gfCNCPoint1[27602] = {X 121.2453, Y 41.6137, Z -2.1667, A 0.000, B 0.000, C 0.000 }
gfCNCPoint1[27603] = {X 121.7141, Y 42.3988, Z -2.1667, A 0.000, B 0.000, C 0.000 }
gfCNCPoint1[27604] = {X 122.0072, Y 43.2649, Z -2.1667, A 0.000, B 0.000, C 0.000 }
gfCNCPoint1[27605] = {X 122.1114, Y 44.1734, Z -2.1667, A 0.000, B 0.000, C 0.000 }
gfCNCPoint1[27606] = {X 122.1116, Y 45.0000, Z -2.1667, A 0.000, B 0.000, C 0.000 }
gfCNCPoint1[27607] = {X 122.0033, Y 45.9613, Z -2.1667, A 0.000, B 0.000, C 0.000 }
gfCNCPoint1[27608] = {X 121.6838, Y 46.8744, Z -2.1667, A 0.000, B 0.000, C 0.000 }
gfCNCPoint1[27609] = {X 121.1691, Y 47.6935, Z -2.1667, A 0.000, B 0.000, C 0.000 }
gfCNCPoint1[27610] = {X 120.4850, Y 48.3775, Z -2.1667, A 0.000, B 0.000, C 0.000 }
gfCNCPoint1[27611] = {X 119.6660, Y 48.8922, Z -2.1667, A 0.000, B 0.000, C 0.000 }
gfCNCPoint1[27612] = {X 118.7529, Y 49.2117, Z -2.1667, A 0.000, B 0.000, C 0.000 }
gfCNCPoint1[27613] = {X 117.7916, Y 49.3200, Z -2.1667, A 0.000, B 0.000, C 0.000 }
gfCNCPoint1[27614] = {X 111.9185, Y 49.3200, Z -2.1667, A 0.000, B 0.000, C 0.000 }
gfCNCPoint1[27615] = {X 110.9619, Y 49.2128, Z -2.1667, A 0.000, B 0.000, C 0.000 }
gfCNCPoint1[27616] = {X 110.0529, Y 48.8964, Z -2.1667, A 0.000, B 0.000, C 0.000 }
gfCNCPoint1[27617] = {X 109.2365, Y 48.3866, Z -2.1667, A 0.000, B 0.000, C 0.000 }
gfCNCPoint1[27618] = {X 108.5532, Y 47.7087, Z -2.1667, A 0.000, B 0.000, C 0.000 }
gfCNCPoint1[27619] = {X 108.0369, Y 46.8963, Z -2.1667, A 0.000, B 0.000, C 0.000 }
gfCNCPoint1[27620] = {X 107.7134, Y 45.9898, Z -2.1667, A 0.000, B 0.000, C 0.000 }
gfCNCPoint1[27621] = {X 107.5986, Y 45.0341, Z -2.1667, A 0.000, B 0.000, C 0.000 }
gfCNCPoint1[27622] = {X 107.5985, Y 44.1778, Z -2.1667, A 0.000, B 0.000, C 0.000 }
gfCNCPoint1[27623] = {X 107.6341, Y 43.6353, Z -2.1667, A 0.000, B 0.000, C 0.000 }
gfCNCPoint1[27624] = {X 107.7405, Y 43.1023, Z -2.1667, A 0.000, B 0.000, C 0.000 }
gfCNCPoint1[27625] = {X 107.9071, Y 42.6088, Z -2.1667, A 0.000, B 0.000, C 0.000 }
gfCNCPoint1[27626] = {X 108.1343, Y 42.1400, Z -2.1667, A 0.000, B 0.000, C 0.000 }
gfCNCPoint1[27627] = {X 108.5859, Y 41.4664, Z -2.1667, A 0.000, B 0.000, C 0.000 }
gfCNCPoint1[27628] = {X 109.1269, Y 40.8623, Z -2.1667, A 0.000, B 0.000, C 0.000 }
gfCNCPoint1[27629] = {X 109.1268, Y 39.2937, Z -2.1667, A 0.000, B 0.000, C 0.000 }
gfCNCPoint1[27630] = {X 106.1118, Y 46.6615, Z -2.1667, A 0.000, B 0.000, C 0.000 }
gfCNCPoint1[27631] = {X 105.7417, Y 47.3611, Z -2.1667, A 0.000, B 0.000, C 0.000 }
gfCNCPoint1[27632] = {X 105.2502, Y 47.9815, Z -2.1667, A 0.000, B 0.000, C 0.000 }
gfCNCPoint1[27633] = {X 104.6538, Y 48.5018, Z -2.1667, A 0.000, B 0.000, C 0.000 }
gfCNCPoint1[27634] = {X 103.9724, Y 48.9046, Z -2.1667, A 0.000, B 0.000, C 0.000 }
gfCNCPoint1[27635] = {X 103.0287, Y 49.2242, Z -2.1667, A 0.000, B 0.000, C 0.000 }
gfCNCPoint1[27636] = {X 102.0368, Y 49.3191, Z -2.1667, A 0.000, B 0.000, C 0.000 }
gfCNCPoint1[27637] = {X 101.0496, Y 49.1842, Z -2.1667, A 0.000, B 0.000, C 0.000 }
gfCNCPoint1[27638] = {X 100.1195, Y 48.8268, Z -2.1667, A 0.000, B 0.000, C 0.000 }
gfCNCPoint1[27639] = {X 99.2961, Y 48.2657, Z -2.1667, A 0.000, B 0.000, C 0.000 }
gfCNCPoint1[27640] = {X 98.6231, Y 47.5309, Z -2.1667, A 0.000, B 0.000, C 0.000 }
gfCNCPoint1[27641] = {X 98.1363, Y 46.6615, Z -2.1667, A 0.000, B 0.000, C 0.000 }
gfCNCPoint1[27642] = {X 95.1301, Y 39.3093, Z -2.1667, A 0.000, B 0.000, C 0.000 }
gfCNCPoint1[27643] = {X 95.1302, Y 40.9055, Z -2.1667, A 0.000, B 0.000, C 0.000 }
gfCNCPoint1[27644] = {X 95.6600, Y 41.4488, Z -2.1667, A 0.000, B 0.000, C 0.000 }
gfCNCPoint1[27645] = {X 96.0887, Y 42.0749, Z -2.1667, A 0.000, B 0.000, C 0.000 }
gfCNCPoint1[27646] = {X 96.3308, Y 42.5747, Z -2.1667, A 0.000, B 0.000, C 0.000 }
gfCNCPoint1[27647] = {X 96.5082, Y 43.1009, Z -2.1667, A 0.000, B 0.000, C 0.000 }
gfCNCPoint1[27648] = {X 96.6185, Y 43.6488, Z -2.1667, A 0.000, B 0.000, C 0.000 }
gfCNCPoint1[27649] = {X 96.6585, Y 44.2063, Z -2.1667, A 0.000, B 0.000, C 0.000 }
gfCNCPoint1[27650] = {X 96.6583, Y 45.0415, Z -2.1667, A 0.000, B 0.000, C 0.000 }
gfCNCPoint1[27651] = {X 96.5422, Y 45.9960, Z -2.1667, A 0.000, B 0.000, C 0.000 }
gfCNCPoint1[27652] = {X 96.2178, Y 46.9011, Z -2.1667, A 0.000, B 0.000, C 0.000 }
gfCNCPoint1[27653] = {X 95.7012, Y 47.7120, Z -2.1667, A 0.000, B 0.000, C 0.000 }
gfCNCPoint1[27654] = {X 95.0181, Y 48.3886, Z -2.1667, A 0.000, B 0.000, C 0.000 }
gfCNCPoint1[27655] = {X 94.2022, Y 48.8973, Z -2.1667, A 0.000, B 0.000, C 0.000 }
gfCNCPoint1[27656] = {X 93.2940, Y 49.2130, Z -2.1667, A 0.000, B 0.000, C 0.000 }
gfCNCPoint1[27657] = {X 92.3385, Y 49.3200, Z -2.1667, A 0.000, B 0.000, C 0.000 }
gfCNCPoint1[27658] = {X 85.8951, Y 49.3200, Z -2.1667, A 0.000, B 0.000, C 0.000 }
gfCNCPoint1[27659] = {X 84.9387, Y 49.2128, Z -2.1667, A 0.000, B 0.000, C 0.000 }
gfCNCPoint1[27660] = {X 84.0297, Y 48.8965, Z -2.1667, A 0.000, B 0.000, C 0.000 }
gfCNCPoint1[27661] = {X 83.2134, Y 48.3869, Z -2.1667, A 0.000, B 0.000, C 0.000 }
gfCNCPoint1[27662] = {X 82.5301, Y 47.7091, Z -2.1667, A 0.000, B 0.000, C 0.000 }
gfCNCPoint1[27663] = {X 82.0138, Y 46.8970, Z -2.1667, A 0.000, B 0.000, C 0.000 }
gfCNCPoint1[27664] = {X 81.6902, Y 45.9906, Z -2.1667, A 0.000, B 0.000, C 0.000 }
gfCNCPoint1[27665] = {X 81.5752, Y 45.0351, Z -2.1667, A 0.000, B 0.000, C 0.000 }
gfCNCPoint1[27666] = {X 81.5751, Y 44.2068, Z -2.1667, A 0.000, B 0.000, C 0.000 }
gfCNCPoint1[27667] = {X 81.6809, Y 43.2777, Z -2.1667, A 0.000, B 0.000, C 0.000 }
gfCNCPoint1[27668] = {X 81.9815, Y 42.3922, Z -2.1667, A 0.000, B 0.000, C 0.000 }
gfCNCPoint1[27669] = {X 82.4630, Y 41.5906, Z -2.1667, A 0.000, B 0.000, C 0.000 }
gfCNCPoint1[27670] = {X 83.1037, Y 40.9095, Z -2.1667, A 0.000, B 0.000, C 0.000 }
gfCNCPoint1[27671] = {X 83.1036, Y 28.5922, Z -2.1667, A 0.000, B 0.000, C 0.000 }
gfCNCPoint1[27672] = {X 79.1036, Y 28.5922, Z -2.1667, A 0.000, B 0.000, C 0.000 }
gfCNCPoint1[27673] = {X 83.1836, Y 28.5922, Z -2.1667, A 0.000, B 0.000, C 0.000 }
gfCNCPoint1[27674] = {X 83.1834, Y 16.2375, Z -2.1667, A 0.000, B 0.000, C 0.000 }
gfCNCPoint1[27675] = {X 82.5450, Y 15.5770, Z -2.1667, A 0.000, B 0.000, C 0.000 }
gfCNCPoint1[27676] = {X 82.0638, Y 14.7944, Z -2.1667, A 0.000, B 0.000, C 0.000 }
gfCNCPoint1[27677] = {X 81.7625, Y 13.9265, Z -2.1667, A 0.000, B 0.000, C 0.000 }
gfCNCPoint1[27678] = {X 81.6552, Y 13.0142, Z -2.1667, A 0.000, B 0.000, C 0.000 }
gfCNCPoint1[27679] = {X 81.6551, Y 12.1868, Z -2.1667, A 0.000, B 0.000, C 0.000 }
gfCNCPoint1[27680] = {X 81.7614, Y 11.2433, Z -2.1667, A 0.000, B 0.000, C 0.000 }
gfCNCPoint1[27681] = {X 82.0750, Y 10.3472, Z -2.1667, A 0.000, B 0.000, C 0.000 }
gfCNCPoint1[27682] = {X 82.5801, Y 9.5432, Z -2.1667, A 0.000, B 0.000, C 0.000 }
gfCNCPoint1[27683] = {X 83.2515, Y 8.8719, Z -2.1667, A 0.000, B 0.000, C 0.000 }
gfCNCPoint1[27684] = {X 84.0554, Y 8.3667, Z -2.1667, A 0.000, B 0.000, C 0.000 }
gfCNCPoint1[27685] = {X 84.9516, Y 8.0531, Z -2.1667, A 0.000, B 0.000, C 0.000 }
gfCNCPoint1[27686] = {X 85.8951, Y 7.9468, Z -2.1667, A 0.000, B 0.000, C 0.000 }
gfCNCPoint1[27687] = {X 94.0497, Y 7.9468, Z -2.1667, A 0.000, B 0.000, C 0.000 }
gfCNCPoint1[27688] = {X 94.9932, Y 8.0531, Z -2.1667, A 0.000, B 0.000, C 0.000 }
gfCNCPoint1[27689] = {X 95.8893, Y 8.3667, Z -2.1667, A 0.000, B 0.000, C 0.000 }
gfCNCPoint1[27690] = {X 96.6933, Y 8.8718, Z -2.1667, A 0.000, B 0.000, C 0.000 }
gfCNCPoint1[27691] = {X 97.3646, Y 9.5432, Z -2.1667, A 0.000, B 0.000, C 0.000 }
gfCNCPoint1[27692] = {X 97.8698, Y 10.3471, Z -2.1667, A 0.000, B 0.000, C 0.000 }
gfCNCPoint1[27693] = {X 98.1834, Y 11.2433, Z -2.1667, A 0.000, B 0.000, C 0.000 }
gfCNCPoint1[27694] = {X 98.2897, Y 12.1868, Z -2.1667, A 0.000, B 0.000, C 0.000 }
gfCNCPoint1[27695] = {X 98.2897, Y 12.9781, Z -2.1667, A 0.000, B 0.000, C 0.000 }
gfCNCPoint1[27696] = {X 98.2155, Y 13.7669, Z -2.1667, A 0.000, B 0.000, C 0.000 }
gfCNCPoint1[27697] = {X 97.9959, Y 14.5281, Z -2.1667, A 0.000, B 0.000, C 0.000 }
gfCNCPoint1[27698] = {X 97.6385, Y 15.2352, Z -2.1667, A 0.000, B 0.000, C 0.000 }
gfCNCPoint1[27699] = {X 101.8779, Y 25.7443, Z -2.1667, A 0.000, B 0.000, C 0.000 }
gfCNCPoint1[27700] = {X 101.9522, Y 25.5604, Z -2.1667, A 0.000, B 0.000, C 0.000 }
gfCNCPoint1[27701] = {X 106.1061, Y 15.2145, Z -2.1667, A 0.000, B 0.000, C 0.000 }
gfCNCPoint1[27702] = {X 105.7606, Y 14.5250, Z -2.1667, A 0.000, B 0.000, C 0.000 }
gfCNCPoint1[27703] = {X 105.5457, Y 13.7844, Z -2.1667, A 0.000, B 0.000, C 0.000 }
gfCNCPoint1[27704] = {X 105.4685, Y 13.0172, Z -2.1667, A 0.000, B 0.000, C 0.000 }
gfCNCPoint1[27705] = {X 105.4683, Y 12.1868, Z -2.1667, A 0.000, B 0.000, C 0.000 }
gfCNCPoint1[27706] = {X 105.5746, Y 11.2433, Z -2.1667, A 0.000, B 0.000, C 0.000 }
gfCNCPoint1[27707] = {X 105.8882, Y 10.3471, Z -2.1667, A 0.000, B 0.000, C 0.000 }
gfCNCPoint1[27708] = {X 106.3933, Y 9.5432, Z -2.1667, A 0.000, B 0.000, C 0.000 }
gfCNCPoint1[27709] = {X 107.0647, Y 8.8718, Z -2.1667, A 0.000, B 0.000, C 0.000 }
gfCNCPoint1[27710] = {X 107.8686, Y 8.3667, Z -2.1667, A 0.000, B 0.000, C 0.000 }
gfCNCPoint1[27711] = {X 108.7648, Y 8.0531, Z -2.1667, A 0.000, B 0.000, C 0.000 }
gfCNCPoint1[27712] = {X 109.7083, Y 7.9468, Z -2.1667, A 0.000, B 0.000, C 0.000 }
gfCNCPoint1[27713] = {X 117.7916, Y 7.9468, Z -2.1667, A 0.000, B 0.000, C 0.000 }
gfCNCPoint1[27714] = {X 118.7351, Y 8.0531, Z -2.1667, A 0.000, B 0.000, C 0.000 }
gfCNCPoint1[27715] = {X 119.6312, Y 8.3667, Z -2.1667, A 0.000, B 0.000, C 0.000 }
gfCNCPoint1[27716] = {X 120.4352, Y 8.8718, Z -2.1667, A 0.000, B 0.000, C 0.000 }
gfCNCPoint1[27717] = {X 121.1065, Y 9.5432, Z -2.1667, A 0.000, B 0.000, C 0.000 }
gfCNCPoint1[27718] = {X 121.6117, Y 10.3471, Z -2.1667, A 0.000, B 0.000, C 0.000 }
gfCNCPoint1[27719] = {X 121.9253, Y 11.2433, Z -2.1667, A 0.000, B 0.000, C 0.000 }
gfCNCPoint1[27720] = {X 122.0316, Y 12.1868, Z -2.1667, A 0.000, B 0.000, C 0.000 }
gfCNCPoint1[27721] = {X 122.0316, Y 12.9781, Z -2.1667, A 0.000, B 0.000, C 0.000 }
gfCNCPoint1[27722] = {X 121.9302, Y 13.8998, Z -2.1667, A 0.000, B 0.000, C 0.000 }
gfCNCPoint1[27723] = {X 121.6308, Y 14.7774, Z -2.1667, A 0.000, B 0.000, C 0.000 }
gfCNCPoint1[27724] = {X 121.1479, Y 15.5690, Z -2.1667, A 0.000, B 0.000, C 0.000 }
gfCNCPoint1[27725] = {X 120.5044, Y 16.2366, Z -2.1667, A 0.000, B 0.000, C 0.000 }
gfCNCPoint1[27726] = {X 120.5031, Y 40.9518, Z -2.1667, A 0.000, B 0.000, C 0.000 }
gfCNCPoint1[27727] = {X 120.5703, Y 41.0062, Z -2.1667, A 0.000, B 0.000, C 0.000 }
gfCNCPoint1[27728] = {X 121.1819, Y 41.6626, Z -2.1667, A 0.000, B 0.000, C 0.000 }
gfCNCPoint1[27729] = {X 121.6417, Y 42.4329, Z -2.1667, A 0.000, B 0.000, C 0.000 }
gfCNCPoint1[27730] = {X 121.9292, Y 43.2827, Z -2.1667, A 0.000, B 0.000, C 0.000 }
gfCNCPoint1[27731] = {X 122.0314, Y 44.1740, Z -2.1667, A 0.000, B 0.000, C 0.000 }
gfCNCPoint1[27732] = {X 122.0316, Y 45.0000, Z -2.1667, A 0.000, B 0.000, C 0.000 }
gfCNCPoint1[27733] = {X 121.9253, Y 45.9435, Z -2.1667, A 0.000, B 0.000, C 0.000 }
gfCNCPoint1[27734] = {X 121.6117, Y 46.8397, Z -2.1667, A 0.000, B 0.000, C 0.000 }
gfCNCPoint1[27735] = {X 121.1065, Y 47.6436, Z -2.1667, A 0.000, B 0.000, C 0.000 }
gfCNCPoint1[27736] = {X 120.4352, Y 48.3150, Z -2.1667, A 0.000, B 0.000, C 0.000 }
gfCNCPoint1[27737] = {X 119.6312, Y 48.8201, Z -2.1667, A 0.000, B 0.000, C 0.000 }
gfCNCPoint1[27738] = {X 118.7351, Y 49.1337, Z -2.1667, A 0.000, B 0.000, C 0.000 }
gfCNCPoint1[27739] = {X 117.7916, Y 49.2400, Z -2.1667, A 0.000, B 0.000, C 0.000 }
gfCNCPoint1[27740] = {X 111.9185, Y 49.2400, Z -2.1667, A 0.000, B 0.000, C 0.000 }
gfCNCPoint1[27741] = {X 110.9797, Y 49.1348, Z -2.1667, A 0.000, B 0.000, C 0.000 }
gfCNCPoint1[27742] = {X 110.0874, Y 48.8242, Z -2.1667, A 0.000, B 0.000, C 0.000 }
gfCNCPoint1[27743] = {X 109.2861, Y 48.3239, Z -2.1667, A 0.000, B 0.000, C 0.000 }
gfCNCPoint1[27744] = {X 108.6155, Y 47.6585, Z -2.1667, A 0.000, B 0.000, C 0.000 }
gfCNCPoint1[27745] = {X 108.1088, Y 46.8612, Z -2.1667, A 0.000, B 0.000, C 0.000 }
gfCNCPoint1[27746] = {X 107.7913, Y 45.9714, Z -2.1667, A 0.000, B 0.000, C 0.000 }
gfCNCPoint1[27747] = {X 107.6786, Y 45.0335, Z -2.1667, A 0.000, B 0.000, C 0.000 }
gfCNCPoint1[27748] = {X 107.6785, Y 44.1778, Z -2.1667, A 0.000, B 0.000, C 0.000 }
gfCNCPoint1[27749] = {X 107.7135, Y 43.6458, Z -2.1667, A 0.000, B 0.000, C 0.000 }
gfCNCPoint1[27750] = {X 107.8178, Y 43.1230, Z -2.1667, A 0.000, B 0.000, C 0.000 }
gfCNCPoint1[27751] = {X 107.9811, Y 42.6391, Z -2.1667, A 0.000, B 0.000, C 0.000 }
gfCNCPoint1[27752] = {X 108.2039, Y 42.1794, Z -2.1667, A 0.000, B 0.000, C 0.000 }
gfCNCPoint1[27753] = {X 108.6596, Y 41.5020, Z -2.1667, A 0.000, B 0.000, C 0.000 }
gfCNCPoint1[27754] = {X 109.2069, Y 40.8962, Z -2.1667, A 0.000, B 0.000, C 0.000 }
gfCNCPoint1[27755] = {X 109.2068, Y 39.1629, Z -2.1667, A 0.000, B 0.000, C 0.000 }
gfCNCPoint1[27756] = {X 109.0939, Y 39.1629, Z -2.1667, A 0.000, B 0.000, C 0.000 }
gfCNCPoint1[27757] = {X 106.0379, Y 46.6307, Z -2.1667, A 0.000, B 0.000, C 0.000 }
gfCNCPoint1[27758] = {X 105.6747, Y 47.3174, Z -2.1667, A 0.000, B 0.000, C 0.000 }
gfCNCPoint1[27759] = {X 105.1923, Y 47.9263, Z -2.1667, A 0.000, B 0.000, C 0.000 }
gfCNCPoint1[27760] = {X 104.6069, Y 48.4370, Z -2.1667, A 0.000, B 0.000, C 0.000 }
gfCNCPoint1[27761] = {X 103.9382, Y 48.8323, Z -2.1667, A 0.000, B 0.000, C 0.000 }
gfCNCPoint1[27762] = {X 103.0119, Y 49.1460, Z -2.1667, A 0.000, B 0.000, C 0.000 }
gfCNCPoint1[27763] = {X 102.0384, Y 49.2391, Z -2.1667, A 0.000, B 0.000, C 0.000 }
gfCNCPoint1[27764] = {X 101.0695, Y 49.1068, Z -2.1667, A 0.000, B 0.000, C 0.000 }
gfCNCPoint1[27765] = {X 100.1566, Y 48.7559, Z -2.1667, A 0.000, B 0.000, C 0.000 }
gfCNCPoint1[27766] = {X 99.3484, Y 48.2052, Z -2.1667, A 0.000, B 0.000, C 0.000 }
gfCNCPoint1[27767] = {X 98.6879, Y 47.4840, Z -2.1667, A 0.000, B 0.000, C 0.000 }
gfCNCPoint1[27768] = {X 98.2102, Y 46.6307, Z -2.1667, A 0.000, B 0.000, C 0.000 }
gfCNCPoint1[27769] = {X 95.0500, Y 38.9022, Z -2.1667, A 0.000, B 0.000, C 0.000 }
gfCNCPoint1[27770] = {X 95.0502, Y 40.9423, Z -2.1667, A 0.000, B 0.000, C 0.000 }
gfCNCPoint1[27771] = {X 95.5865, Y 41.4854, Z -2.1667, A 0.000, B 0.000, C 0.000 }
gfCNCPoint1[27772] = {X 96.0190, Y 42.1142, Z -2.1667, A 0.000, B 0.000, C 0.000 }
gfCNCPoint1[27773] = {X 96.2568, Y 42.6049, Z -2.1667, A 0.000, B 0.000, C 0.000 }
gfCNCPoint1[27774] = {X 96.4309, Y 43.1216, Z -2.1667, A 0.000, B 0.000, C 0.000 }
gfCNCPoint1[27775] = {X 96.5392, Y 43.6596, Z -2.1667, A 0.000, B 0.000, C 0.000 }
gfCNCPoint1[27776] = {X 96.5785, Y 44.2069, Z -2.1667, A 0.000, B 0.000, C 0.000 }
gfCNCPoint1[27777] = {X 96.5783, Y 45.0408, Z -2.1667, A 0.000, B 0.000, C 0.000 }
gfCNCPoint1[27778] = {X 96.4643, Y 45.9775, Z -2.1667, A 0.000, B 0.000, C 0.000 }
gfCNCPoint1[27779] = {X 96.1459, Y 46.8659, Z -2.1667, A 0.000, B 0.000, C 0.000 }
gfCNCPoint1[27780] = {X 95.6389, Y 47.6618, Z -2.1667, A 0.000, B 0.000, C 0.000 }
gfCNCPoint1[27781] = {X 94.9685, Y 48.3258, Z -2.1667, A 0.000, B 0.000, C 0.000 }
gfCNCPoint1[27782] = {X 94.1677, Y 48.8251, Z -2.1667, A 0.000, B 0.000, C 0.000 }
gfCNCPoint1[27783] = {X 93.2764, Y 49.1350, Z -2.1667, A 0.000, B 0.000, C 0.000 }
gfCNCPoint1[27784] = {X 92.3385, Y 49.2400, Z -2.1667, A 0.000, B 0.000, C 0.000 }
gfCNCPoint1[27785] = {X 85.8951, Y 49.2400, Z -2.1667, A 0.000, B 0.000, C 0.000 }
gfCNCPoint1[27786] = {X 84.9564, Y 49.1348, Z -2.1667, A 0.000, B 0.000, C 0.000 }
gfCNCPoint1[27787] = {X 84.0643, Y 48.8244, Z -2.1667, A 0.000, B 0.000, C 0.000 }
gfCNCPoint1[27788] = {X 83.2631, Y 48.3242, Z -2.1667, A 0.000, B 0.000, C 0.000 }
gfCNCPoint1[27789] = {X 82.5924, Y 47.6590, Z -2.1667, A 0.000, B 0.000, C 0.000 }
gfCNCPoint1[27790] = {X 82.0857, Y 46.8618, Z -2.1667, A 0.000, B 0.000, C 0.000 }
gfCNCPoint1[27791] = {X 81.7681, Y 45.9723, Z -2.1667, A 0.000, B 0.000, C 0.000 }
gfCNCPoint1[27792] = {X 81.6552, Y 45.0345, Z -2.1667, A 0.000, B 0.000, C 0.000 }
gfCNCPoint1[27793] = {X 81.6551, Y 44.2073, Z -2.1667, A 0.000, B 0.000, C 0.000 }
gfCNCPoint1[27794] = {X 81.7610, Y 43.2863, Z -2.1667, A 0.000, B 0.000, C 0.000 }
gfCNCPoint1[27795] = {X 82.0618, Y 42.4093, Z -2.1667, A 0.000, B 0.000, C 0.000 }
gfCNCPoint1[27796] = {X 82.5435, Y 41.6171, Z -2.1667, A 0.000, B 0.000, C 0.000 }
gfCNCPoint1[27797] = {X 83.1837, Y 40.9465, Z -2.1667, A 0.000, B 0.000, C 0.000 }
gfCNCPoint1[27798] = {X 83.1836, Y 28.5922, Z -2.1667, A 0.000, B 0.000, C 0.000 }
gfCNCPoint1[27799] = {X 79.1836, Y 28.5922, Z -2.1667, A 0.000, B 0.000, C 0.000 }
gfCNCPoint1[27800] = {X 83.2636, Y 28.5922, Z -2.1667, A 0.000, B 0.000, C 0.000 }
gfCNCPoint1[27801] = {X 83.2634, Y 16.1998, Z -2.1667, A 0.000, B 0.000, C 0.000 }
gfCNCPoint1[27802] = {X 82.6255, Y 15.5500, Z -2.1667, A 0.000, B 0.000, C 0.000 }
gfCNCPoint1[27803] = {X 82.1442, Y 14.7770, Z -2.1667, A 0.000, B 0.000, C 0.000 }
gfCNCPoint1[27804] = {X 81.8426, Y 13.9177, Z -2.1667, A 0.000, B 0.000, C 0.000 }
gfCNCPoint1[27805] = {X 81.7352, Y 13.0135, Z -2.1667, A 0.000, B 0.000, C 0.000 }
gfCNCPoint1[27806] = {X 81.7351, Y 12.1868, Z -2.1667, A 0.000, B 0.000, C 0.000 }
gfCNCPoint1[27807] = {X 81.8394, Y 11.2611, Z -2.1667, A 0.000, B 0.000, C 0.000 }
gfCNCPoint1[27808] = {X 82.1470, Y 10.3819, Z -2.1667, A 0.000, B 0.000, C 0.000 }
gfCNCPoint1[27809] = {X 82.6427, Y 9.5931, Z -2.1667, A 0.000, B 0.000, C 0.000 }
gfCNCPoint1[27810] = {X 83.3014, Y 8.9344, Z -2.1667, A 0.000, B 0.000, C 0.000 }
gfCNCPoint1[27811] = {X 84.0901, Y 8.4388, Z -2.1667, A 0.000, B 0.000, C 0.000 }
gfCNCPoint1[27812] = {X 84.9694, Y 8.1311, Z -2.1667, A 0.000, B 0.000, C 0.000 }
gfCNCPoint1[27813] = {X 85.8951, Y 8.0268, Z -2.1667, A 0.000, B 0.000, C 0.000 }
gfCNCPoint1[27814] = {X 94.0497, Y 8.0268, Z -2.1667, A 0.000, B 0.000, C 0.000 }
gfCNCPoint1[27815] = {X 94.9754, Y 8.1311, Z -2.1667, A 0.000, B 0.000, C 0.000 }
gfCNCPoint1[27816] = {X 95.8546, Y 8.4388, Z -2.1667, A 0.000, B 0.000, C 0.000 }
gfCNCPoint1[27817] = {X 96.6434, Y 8.9344, Z -2.1667, A 0.000, B 0.000, C 0.000 }
gfCNCPoint1[27818] = {X 97.3021, Y 9.5931, Z -2.1667, A 0.000, B 0.000, C 0.000 }
gfCNCPoint1[27819] = {X 97.7977, Y 10.3819, Z -2.1667, A 0.000, B 0.000, C 0.000 }
gfCNCPoint1[27820] = {X 98.1054, Y 11.2611, Z -2.1667, A 0.000, B 0.000, C 0.000 }
gfCNCPoint1[27821] = {X 98.2097, Y 12.1868, Z -2.1667, A 0.000, B 0.000, C 0.000 }
gfCNCPoint1[27822] = {X 98.2097, Y 12.9781, Z -2.1667, A 0.000, B 0.000, C 0.000 }
gfCNCPoint1[27823] = {X 98.1343, Y 13.7662, Z -2.1667, A 0.000, B 0.000, C 0.000 }
gfCNCPoint1[27824] = {X 97.9110, Y 14.5258, Z -2.1667, A 0.000, B 0.000, C 0.000 }
gfCNCPoint1[27825] = {X 97.5479, Y 15.2293, Z -2.1667, A 0.000, B 0.000, C 0.000 }
gfCNCPoint1[27826] = {X 101.8774, Y 25.9567, Z -2.1667, A 0.000, B 0.000, C 0.000 }
gfCNCPoint1[27827] = {X 101.9789, Y 25.7088, Z -2.1667, A 0.000, B 0.000, C 0.000 }
gfCNCPoint1[27828] = {X 106.1955, Y 15.2064, Z -2.1667, A 0.000, B 0.000, C 0.000 }
gfCNCPoint1[27829] = {X 105.8450, Y 14.5209, Z -2.1667, A 0.000, B 0.000, C 0.000 }
gfCNCPoint1[27830] = {X 105.6268, Y 13.7824, Z -2.1667, A 0.000, B 0.000, C 0.000 }
gfCNCPoint1[27831] = {X 105.5485, Y 13.0164, Z -2.1667, A 0.000, B 0.000, C 0.000 }
gfCNCPoint1[27832] = {X 105.5483, Y 12.1868, Z -2.1667, A 0.000, B 0.000, C 0.000 }
gfCNCPoint1[27833] = {X 105.6526, Y 11.2611, Z -2.1667, A 0.000, B 0.000, C 0.000 }
gfCNCPoint1[27834] = {X 105.9602, Y 10.3819, Z -2.1667, A 0.000, B 0.000, C 0.000 }
gfCNCPoint1[27835] = {X 106.4559, Y 9.5931, Z -2.1667, A 0.000, B 0.000, C 0.000 }
gfCNCPoint1[27836] = {X 107.1146, Y 8.9344, Z -2.1667, A 0.000, B 0.000, C 0.000 }
gfCNCPoint1[27837] = {X 107.9033, Y 8.4388, Z -2.1667, A 0.000, B 0.000, C 0.000 }
gfCNCPoint1[27838] = {X 108.7826, Y 8.1311, Z -2.1667, A 0.000, B 0.000, C 0.000 }
gfCNCPoint1[27839] = {X 109.7083, Y 8.0268, Z -2.1667, A 0.000, B 0.000, C 0.000 }
gfCNCPoint1[27840] = {X 117.7916, Y 8.0268, Z -2.1667, A 0.000, B 0.000, C 0.000 }
gfCNCPoint1[27841] = {X 118.7173, Y 8.1311, Z -2.1667, A 0.000, B 0.000, C 0.000 }
gfCNCPoint1[27842] = {X 119.5965, Y 8.4388, Z -2.1667, A 0.000, B 0.000, C 0.000 }
gfCNCPoint1[27843] = {X 120.3853, Y 8.9344, Z -2.1667, A 0.000, B 0.000, C 0.000 }
gfCNCPoint1[27844] = {X 121.0440, Y 9.5931, Z -2.1667, A 0.000, B 0.000, C 0.000 }
gfCNCPoint1[27845] = {X 121.5396, Y 10.3819, Z -2.1667, A 0.000, B 0.000, C 0.000 }
gfCNCPoint1[27846] = {X 121.8473, Y 11.2611, Z -2.1667, A 0.000, B 0.000, C 0.000 }
gfCNCPoint1[27847] = {X 121.9516, Y 12.1868, Z -2.1667, A 0.000, B 0.000, C 0.000 }
gfCNCPoint1[27848] = {X 121.9516, Y 12.9781, Z -2.1667, A 0.000, B 0.000, C 0.000 }
gfCNCPoint1[27849] = {X 121.8500, Y 13.8915, Z -2.1667, A 0.000, B 0.000, C 0.000 }
gfCNCPoint1[27850] = {X 121.5504, Y 14.7604, Z -2.1667, A 0.000, B 0.000, C 0.000 }
gfCNCPoint1[27851] = {X 121.0673, Y 15.5422, Z -2.1667, A 0.000, B 0.000, C 0.000 }
gfCNCPoint1[27852] = {X 120.4244, Y 16.1989, Z -2.1667, A 0.000, B 0.000, C 0.000 }
gfCNCPoint1[27853] = {X 120.4231, Y 40.9900, Z -2.1667, A 0.000, B 0.000, C 0.000 }
gfCNCPoint1[27854] = {X 120.5189, Y 41.0675, Z -2.1667, A 0.000, B 0.000, C 0.000 }
gfCNCPoint1[27855] = {X 121.1185, Y 41.7114, Z -2.1667, A 0.000, B 0.000, C 0.000 }
gfCNCPoint1[27856] = {X 121.5694, Y 42.4670, Z -2.1667, A 0.000, B 0.000, C 0.000 }
gfCNCPoint1[27857] = {X 121.8512, Y 43.3005, Z -2.1667, A 0.000, B 0.000, C 0.000 }
gfCNCPoint1[27858] = {X 121.9514, Y 44.1747, Z -2.1667, A 0.000, B 0.000, C 0.000 }
gfCNCPoint1[27859] = {X 121.9516, Y 45.0000, Z -2.1667, A 0.000, B 0.000, C 0.000 }
gfCNCPoint1[27860] = {X 121.8473, Y 45.9257, Z -2.1667, A 0.000, B 0.000, C 0.000 }
gfCNCPoint1[27861] = {X 121.5396, Y 46.8050, Z -2.1667, A 0.000, B 0.000, C 0.000 }
gfCNCPoint1[27862] = {X 121.0440, Y 47.5937, Z -2.1667, A 0.000, B 0.000, C 0.000 }
gfCNCPoint1[27863] = {X 120.3853, Y 48.2524, Z -2.1667, A 0.000, B 0.000, C 0.000 }
gfCNCPoint1[27864] = {X 119.5965, Y 48.7480, Z -2.1667, A 0.000, B 0.000, C 0.000 }
gfCNCPoint1[27865] = {X 118.7173, Y 49.0557, Z -2.1667, A 0.000, B 0.000, C 0.000 }
gfCNCPoint1[27866] = {X 117.7916, Y 49.1600, Z -2.1667, A 0.000, B 0.000, C 0.000 }
gfCNCPoint1[27867] = {X 111.9185, Y 49.1600, Z -2.1667, A 0.000, B 0.000, C 0.000 }
gfCNCPoint1[27868] = {X 110.9974, Y 49.0567, Z -2.1667, A 0.000, B 0.000, C 0.000 }
gfCNCPoint1[27869] = {X 110.1220, Y 48.7521, Z -2.1667, A 0.000, B 0.000, C 0.000 }
gfCNCPoint1[27870] = {X 109.3358, Y 48.2612, Z -2.1667, A 0.000, B 0.000, C 0.000 }
gfCNCPoint1[27871] = {X 108.6778, Y 47.6084, Z -2.1667, A 0.000, B 0.000, C 0.000 }
gfCNCPoint1[27872] = {X 108.1807, Y 46.8261, Z -2.1667, A 0.000, B 0.000, C 0.000 }
gfCNCPoint1[27873] = {X 107.8691, Y 45.9531, Z -2.1667, A 0.000, B 0.000, C 0.000 }
gfCNCPoint1[27874] = {X 107.7586, Y 45.0328, Z -2.1667, A 0.000, B 0.000, C 0.000 }
gfCNCPoint1[27875] = {X 107.7585, Y 44.1778, Z -2.1667, A 0.000, B 0.000, C 0.000 }
gfCNCPoint1[27876] = {X 107.7928, Y 43.6563, Z -2.1667, A 0.000, B 0.000, C 0.000 }
gfCNCPoint1[27877] = {X 107.8950, Y 43.1438, Z -2.1667, A 0.000, B 0.000, C 0.000 }
gfCNCPoint1[27878] = {X 108.0552, Y 42.6694, Z -2.1667, A 0.000, B 0.000, C 0.000 }
gfCNCPoint1[27879] = {X 108.2736, Y 42.2187, Z -2.1667, A 0.000, B 0.000, C 0.000 }
gfCNCPoint1[27880] = {X 108.7333, Y 41.5377, Z -2.1667, A 0.000, B 0.000, C 0.000 }
gfCNCPoint1[27881] = {X 109.2869, Y 40.9305, Z -2.1667, A 0.000, B 0.000, C 0.000 }
gfCNCPoint1[27882] = {X 109.2868, Y 39.0829, Z -2.1667, A 0.000, B 0.000, C 0.000 }
gfCNCPoint1[27883] = {X 109.0402, Y 39.0829, Z -2.1667, A 0.000, B 0.000, C 0.000 }
gfCNCPoint1[27884] = {X 105.9641, Y 46.5999, Z -2.1667, A 0.000, B 0.000, C 0.000 }
gfCNCPoint1[27885] = {X 105.6077, Y 47.2737, Z -2.1667, A 0.000, B 0.000, C 0.000 }
gfCNCPoint1[27886] = {X 105.1344, Y 47.8711, Z -2.1667, A 0.000, B 0.000, C 0.000 }
gfCNCPoint1[27887] = {X 104.5601, Y 48.3721, Z -2.1667, A 0.000, B 0.000, C 0.000 }
gfCNCPoint1[27888] = {X 103.9040, Y 48.7600, Z -2.1667, A 0.000, B 0.000, C 0.000 }
gfCNCPoint1[27889] = {X 102.9952, Y 49.0678, Z -2.1667, A 0.000, B 0.000, C 0.000 }
gfCNCPoint1[27890] = {X 102.0400, Y 49.1592, Z -2.1667, A 0.000, B 0.000, C 0.000 }
gfCNCPoint1[27891] = {X 101.0894, Y 49.0293, Z -2.1667, A 0.000, B 0.000, C 0.000 }
gfCNCPoint1[27892] = {X 100.1937, Y 48.6850, Z -2.1667, A 0.000, B 0.000, C 0.000 }
gfCNCPoint1[27893] = {X 99.4008, Y 48.1448, Z -2.1667, A 0.000, B 0.000, C 0.000 }
gfCNCPoint1[27894] = {X 98.7527, Y 47.4372, Z -2.1667, A 0.000, B 0.000, C 0.000 }
gfCNCPoint1[27895] = {X 98.2840, Y 46.5999, Z -2.1667, A 0.000, B 0.000, C 0.000 }
gfCNCPoint1[27896] = {X 94.9700, Y 38.4951, Z -2.1667, A 0.000, B 0.000, C 0.000 }
gfCNCPoint1[27897] = {X 94.9702, Y 40.9796, Z -2.1667, A 0.000, B 0.000, C 0.000 }
gfCNCPoint1[27898] = {X 95.5130, Y 41.5222, Z -2.1667, A 0.000, B 0.000, C 0.000 }
gfCNCPoint1[27899] = {X 95.9494, Y 42.1536, Z -2.1667, A 0.000, B 0.000, C 0.000 }
gfCNCPoint1[27900] = {X 96.1827, Y 42.6352, Z -2.1667, A 0.000, B 0.000, C 0.000 }
gfCNCPoint1[27901] = {X 96.3537, Y 43.1423, Z -2.1667, A 0.000, B 0.000, C 0.000 }
gfCNCPoint1[27902] = {X 96.4599, Y 43.6704, Z -2.1667, A 0.000, B 0.000, C 0.000 }
gfCNCPoint1[27903] = {X 96.4985, Y 44.2076, Z -2.1667, A 0.000, B 0.000, C 0.000 }
gfCNCPoint1[27904] = {X 96.4983, Y 45.0400, Z -2.1667, A 0.000, B 0.000, C 0.000 }
gfCNCPoint1[27905] = {X 96.3865, Y 45.9591, Z -2.1667, A 0.000, B 0.000, C 0.000 }
gfCNCPoint1[27906] = {X 96.0741, Y 46.8306, Z -2.1667, A 0.000, B 0.000, C 0.000 }
gfCNCPoint1[27907] = {X 95.5767, Y 47.6115, Z -2.1667, A 0.000, B 0.000, C 0.000 }
gfCNCPoint1[27908] = {X 94.9188, Y 48.2631, Z -2.1667, A 0.000, B 0.000, C 0.000 }
gfCNCPoint1[27909] = {X 94.1332, Y 48.7530, Z -2.1667, A 0.000, B 0.000, C 0.000 }
gfCNCPoint1[27910] = {X 93.2587, Y 49.0570, Z -2.1667, A 0.000, B 0.000, C 0.000 }
gfCNCPoint1[27911] = {X 92.3385, Y 49.1600, Z -2.1667, A 0.000, B 0.000, C 0.000 }
gfCNCPoint1[27912] = {X 85.8951, Y 49.1600, Z -2.1667, A 0.000, B 0.000, C 0.000 }
gfCNCPoint1[27913] = {X 84.9741, Y 49.0568, Z -2.1667, A 0.000, B 0.000, C 0.000 }
gfCNCPoint1[27914] = {X 84.0988, Y 48.7522, Z -2.1667, A 0.000, B 0.000, C 0.000 }
gfCNCPoint1[27915] = {X 83.3127, Y 48.2614, Z -2.1667, A 0.000, B 0.000, C 0.000 }
gfCNCPoint1[27916] = {X 82.6547, Y 47.6088, Z -2.1667, A 0.000, B 0.000, C 0.000 }
gfCNCPoint1[27917] = {X 82.1576, Y 46.8267, Z -2.1667, A 0.000, B 0.000, C 0.000 }
gfCNCPoint1[27918] = {X 81.8459, Y 45.9539, Z -2.1667, A 0.000, B 0.000, C 0.000 }
gfCNCPoint1[27919] = {X 81.7352, Y 45.0338, Z -2.1667, A 0.000, B 0.000, C 0.000 }
gfCNCPoint1[27920] = {X 81.7351, Y 44.2079, Z -2.1667, A 0.000, B 0.000, C 0.000 }
gfCNCPoint1[27921] = {X 81.8411, Y 43.2949, Z -2.1667, A 0.000, B 0.000, C 0.000 }
gfCNCPoint1[27922] = {X 82.1421, Y 42.4265, Z -2.1667, A 0.000, B 0.000, C 0.000 }
gfCNCPoint1[27923] = {X 82.6239, Y 41.6438, Z -2.1667, A 0.000, B 0.000, C 0.000 }
gfCNCPoint1[27924] = {X 83.2637, Y 40.9839, Z -2.1667, A 0.000, B 0.000, C 0.000 }
gfCNCPoint1[27925] = {X 83.2636, Y 28.5922, Z -2.1667, A 0.000, B 0.000, C 0.000 }
gfCNCPoint1[27926] = {X 79.2636, Y 28.5922, Z -2.1667, A 0.000, B 0.000, C 0.000 }
gfCNCPoint1[27927] = {X 83.3436, Y 28.5922, Z -2.1667, A 0.000, B 0.000, C 0.000 }
gfCNCPoint1[27928] = {X 83.3434, Y 16.1616, Z -2.1667, A 0.000, B 0.000, C 0.000 }
gfCNCPoint1[27929] = {X 82.7059, Y 15.5228, Z -2.1667, A 0.000, B 0.000, C 0.000 }
gfCNCPoint1[27930] = {X 82.2245, Y 14.7594, Z -2.1667, A 0.000, B 0.000, C 0.000 }
gfCNCPoint1[27931] = {X 81.9227, Y 13.9089, Z -2.1667, A 0.000, B 0.000, C 0.000 }
gfCNCPoint1[27932] = {X 81.8152, Y 13.0128, Z -2.1667, A 0.000, B 0.000, C 0.000 }
gfCNCPoint1[27933] = {X 81.8151, Y 12.1868, Z -2.1667, A 0.000, B 0.000, C 0.000 }
gfCNCPoint1[27934] = {X 81.9174, Y 11.2789, Z -2.1667, A 0.000, B 0.000, C 0.000 }
gfCNCPoint1[27935] = {X 82.2191, Y 10.4166, Z -2.1667, A 0.000, B 0.000, C 0.000 }
gfCNCPoint1[27936] = {X 82.7052, Y 9.6430, Z -2.1667, A 0.000, B 0.000, C 0.000 }
gfCNCPoint1[27937] = {X 83.3512, Y 8.9969, Z -2.1667, A 0.000, B 0.000, C 0.000 }
gfCNCPoint1[27938] = {X 84.1248, Y 8.5109, Z -2.1667, A 0.000, B 0.000, C 0.000 }
gfCNCPoint1[27939] = {X 84.9872, Y 8.2091, Z -2.1667, A 0.000, B 0.000, C 0.000 }
gfCNCPoint1[27940] = {X 85.8951, Y 8.1068, Z -2.1667, A 0.000, B 0.000, C 0.000 }
gfCNCPoint1[27941] = {X 94.0497, Y 8.1068, Z -2.1667, A 0.000, B 0.000, C 0.000 }
gfCNCPoint1[27942] = {X 94.9576, Y 8.2091, Z -2.1667, A 0.000, B 0.000, C 0.000 }
gfCNCPoint1[27943] = {X 95.8199, Y 8.5109, Z -2.1667, A 0.000, B 0.000, C 0.000 }
gfCNCPoint1[27944] = {X 96.5935, Y 8.9969, Z -2.1667, A 0.000, B 0.000, C 0.000 }
gfCNCPoint1[27945] = {X 97.2395, Y 9.6430, Z -2.1667, A 0.000, B 0.000, C 0.000 }
gfCNCPoint1[27946] = {X 97.7256, Y 10.4166, Z -2.1667, A 0.000, B 0.000, C 0.000 }
gfCNCPoint1[27947] = {X 98.0274, Y 11.2789, Z -2.1667, A 0.000, B 0.000, C 0.000 }
gfCNCPoint1[27948] = {X 98.1297, Y 12.1868, Z -2.1667, A 0.000, B 0.000, C 0.000 }
gfCNCPoint1[27949] = {X 98.1297, Y 12.9781, Z -2.1667, A 0.000, B 0.000, C 0.000 }
gfCNCPoint1[27950] = {X 98.0630, Y 13.7123, Z -2.1667, A 0.000, B 0.000, C 0.000 }
gfCNCPoint1[27951] = {X 97.8654, Y 14.4225, Z -2.1667, A 0.000, B 0.000, C 0.000 }
gfCNCPoint1[27952] = {X 97.5432, Y 15.0856, Z -2.1667, A 0.000, B 0.000, C 0.000 }
gfCNCPoint1[27953] = {X 97.4969, Y 15.1605, Z -2.1667, A 0.000, B 0.000, C 0.000 }
gfCNCPoint1[27954] = {X 97.4490, Y 15.2344, Z -2.1667, A 0.000, B 0.000, C 0.000 }
gfCNCPoint1[27955] = {X 97.4844, Y 15.2809, Z -2.1667, A 0.000, B 0.000, C 0.000 }
gfCNCPoint1[27956] = {X 101.8768, Y 26.1692, Z -2.1667, A 0.000, B 0.000, C 0.000 }
gfCNCPoint1[27957] = {X 102.0530, Y 25.7388, Z -2.1667, A 0.000, B 0.000, C 0.000 }
gfCNCPoint1[27958] = {X 106.2851, Y 15.1980, Z -2.1667, A 0.000, B 0.000, C 0.000 }
gfCNCPoint1[27959] = {X 106.2417, Y 15.1296, Z -2.1667, A 0.000, B 0.000, C 0.000 }
gfCNCPoint1[27960] = {X 106.1997, Y 15.0605, Z -2.1667, A 0.000, B 0.000, C 0.000 }
gfCNCPoint1[27961] = {X 105.8901, Y 14.4160, Z -2.1667, A 0.000, B 0.000, C 0.000 }
gfCNCPoint1[27962] = {X 105.6977, Y 13.7273, Z -2.1667, A 0.000, B 0.000, C 0.000 }
gfCNCPoint1[27963] = {X 105.6285, Y 13.0157, Z -2.1667, A 0.000, B 0.000, C 0.000 }
gfCNCPoint1[27964] = {X 105.6283, Y 12.1868, Z -2.1667, A 0.000, B 0.000, C 0.000 }
gfCNCPoint1[27965] = {X 105.7306, Y 11.2789, Z -2.1667, A 0.000, B 0.000, C 0.000 }
gfCNCPoint1[27966] = {X 106.0323, Y 10.4166, Z -2.1667, A 0.000, B 0.000, C 0.000 }
gfCNCPoint1[27967] = {X 106.5184, Y 9.6430, Z -2.1667, A 0.000, B 0.000, C 0.000 }
gfCNCPoint1[27968] = {X 107.1644, Y 8.9969, Z -2.1667, A 0.000, B 0.000, C 0.000 }
gfCNCPoint1[27969] = {X 107.9380, Y 8.5109, Z -2.1667, A 0.000, B 0.000, C 0.000 }
gfCNCPoint1[27970] = {X 108.8004, Y 8.2091, Z -2.1667, A 0.000, B 0.000, C 0.000 }
gfCNCPoint1[27971] = {X 109.7083, Y 8.1068, Z -2.1667, A 0.000, B 0.000, C 0.000 }
gfCNCPoint1[27972] = {X 117.7916, Y 8.1068, Z -2.1667, A 0.000, B 0.000, C 0.000 }
gfCNCPoint1[27973] = {X 118.6995, Y 8.2091, Z -2.1667, A 0.000, B 0.000, C 0.000 }
gfCNCPoint1[27974] = {X 119.5618, Y 8.5109, Z -2.1667, A 0.000, B 0.000, C 0.000 }
gfCNCPoint1[27975] = {X 120.3354, Y 8.9969, Z -2.1667, A 0.000, B 0.000, C 0.000 }
gfCNCPoint1[27976] = {X 120.9814, Y 9.6430, Z -2.1667, A 0.000, B 0.000, C 0.000 }
gfCNCPoint1[27977] = {X 121.4675, Y 10.4166, Z -2.1667, A 0.000, B 0.000, C 0.000 }
gfCNCPoint1[27978] = {X 121.7693, Y 11.2789, Z -2.1667, A 0.000, B 0.000, C 0.000 }
gfCNCPoint1[27979] = {X 121.8716, Y 12.1868, Z -2.1667, A 0.000, B 0.000, C 0.000 }
gfCNCPoint1[27980] = {X 121.8716, Y 12.9781, Z -2.1667, A 0.000, B 0.000, C 0.000 }
gfCNCPoint1[27981] = {X 121.7699, Y 13.8832, Z -2.1667, A 0.000, B 0.000, C 0.000 }
gfCNCPoint1[27982] = {X 121.4700, Y 14.7431, Z -2.1667, A 0.000, B 0.000, C 0.000 }
gfCNCPoint1[27983] = {X 120.9868, Y 15.5151, Z -2.1667, A 0.000, B 0.000, C 0.000 }
gfCNCPoint1[27984] = {X 120.3444, Y 16.1607, Z -2.1667, A 0.000, B 0.000, C 0.000 }
gfCNCPoint1[27985] = {X 120.3431, Y 41.0281, Z -2.1667, A 0.000, B 0.000, C 0.000 }
gfCNCPoint1[27986] = {X 120.4674, Y 41.1288, Z -2.1667, A 0.000, B 0.000, C 0.000 }
gfCNCPoint1[27987] = {X 121.0552, Y 41.7602, Z -2.1667, A 0.000, B 0.000, C 0.000 }
gfCNCPoint1[27988] = {X 121.4970, Y 42.5011, Z -2.1667, A 0.000, B 0.000, C 0.000 }
gfCNCPoint1[27989] = {X 121.7732, Y 43.3183, Z -2.1667, A 0.000, B 0.000, C 0.000 }
gfCNCPoint1[27990] = {X 121.8714, Y 44.1754, Z -2.1667, A 0.000, B 0.000, C 0.000 }
gfCNCPoint1[27991] = {X 121.8716, Y 45.0000, Z -2.1667, A 0.000, B 0.000, C 0.000 }
gfCNCPoint1[27992] = {X 121.7693, Y 45.9079, Z -2.1667, A 0.000, B 0.000, C 0.000 }
gfCNCPoint1[27993] = {X 121.4675, Y 46.7702, Z -2.1667, A 0.000, B 0.000, C 0.000 }
gfCNCPoint1[27994] = {X 120.9814, Y 47.5438, Z -2.1667, A 0.000, B 0.000, C 0.000 }
gfCNCPoint1[27995] = {X 120.3354, Y 48.1899, Z -2.1667, A 0.000, B 0.000, C 0.000 }
gfCNCPoint1[27996] = {X 119.5618, Y 48.6760, Z -2.1667, A 0.000, B 0.000, C 0.000 }
gfCNCPoint1[27997] = {X 118.6995, Y 48.9777, Z -2.1667, A 0.000, B 0.000, C 0.000 }
gfCNCPoint1[27998] = {X 117.7916, Y 49.0800, Z -2.1667, A 0.000, B 0.000, C 0.000 }
gfCNCPoint1[27999] = {X 111.9185, Y 49.0800, Z -2.1667, A 0.000, B 0.000, C 0.000 }
gfCNCPoint1[28000] = {X 111.0151, Y 48.9787, Z -2.1667, A 0.000, B 0.000, C 0.000 }
gfCNCPoint1[28001] = {X 110.1565, Y 48.6799, Z -2.1667, A 0.000, B 0.000, C 0.000 }
gfCNCPoint1[28002] = {X 109.3855, Y 48.1985, Z -2.1667, A 0.000, B 0.000, C 0.000 }
gfCNCPoint1[28003] = {X 108.7401, Y 47.5582, Z -2.1667, A 0.000, B 0.000, C 0.000 }
gfCNCPoint1[28004] = {X 108.2526, Y 46.7909, Z -2.1667, A 0.000, B 0.000, C 0.000 }
gfCNCPoint1[28005] = {X 107.9470, Y 45.9348, Z -2.1667, A 0.000, B 0.000, C 0.000 }
gfCNCPoint1[28006] = {X 107.8386, Y 45.0322, Z -2.1667, A 0.000, B 0.000, C 0.000 }
gfCNCPoint1[28007] = {X 107.8385, Y 44.1778, Z -2.1667, A 0.000, B 0.000, C 0.000 }
gfCNCPoint1[28008] = {X 107.8721, Y 43.6668, Z -2.1667, A 0.000, B 0.000, C 0.000 }
gfCNCPoint1[28009] = {X 107.9723, Y 43.1646, Z -2.1667, A 0.000, B 0.000, C 0.000 }
gfCNCPoint1[28010] = {X 108.1292, Y 42.6996, Z -2.1667, A 0.000, B 0.000, C 0.000 }
gfCNCPoint1[28011] = {X 108.3432, Y 42.2581, Z -2.1667, A 0.000, B 0.000, C 0.000 }
gfCNCPoint1[28012] = {X 108.8069, Y 41.5734, Z -2.1667, A 0.000, B 0.000, C 0.000 }
gfCNCPoint1[28013] = {X 109.3669, Y 40.9650, Z -2.1667, A 0.000, B 0.000, C 0.000 }
gfCNCPoint1[28014] = {X 109.3668, Y 39.0029, Z -2.1667, A 0.000, B 0.000, C 0.000 }
gfCNCPoint1[28015] = {X 108.9865, Y 39.0029, Z -2.1667, A 0.000, B 0.000, C 0.000 }
gfCNCPoint1[28016] = {X 105.8902, Y 46.5692, Z -2.1667, A 0.000, B 0.000, C 0.000 }
gfCNCPoint1[28017] = {X 105.5407, Y 47.2300, Z -2.1667, A 0.000, B 0.000, C 0.000 }
gfCNCPoint1[28018] = {X 105.0765, Y 47.8159, Z -2.1667, A 0.000, B 0.000, C 0.000 }
gfCNCPoint1[28019] = {X 104.5133, Y 48.3073, Z -2.1667, A 0.000, B 0.000, C 0.000 }
gfCNCPoint1[28020] = {X 103.8698, Y 48.6877, Z -2.1667, A 0.000, B 0.000, C 0.000 }
gfCNCPoint1[28021] = {X 102.9784, Y 48.9895, Z -2.1667, A 0.000, B 0.000, C 0.000 }
gfCNCPoint1[28022] = {X 102.0417, Y 49.0792, Z -2.1667, A 0.000, B 0.000, C 0.000 }
gfCNCPoint1[28023] = {X 101.1093, Y 48.9518, Z -2.1667, A 0.000, B 0.000, C 0.000 }
gfCNCPoint1[28024] = {X 100.2309, Y 48.6142, Z -2.1667, A 0.000, B 0.000, C 0.000 }
gfCNCPoint1[28025] = {X 99.4532, Y 48.0843, Z -2.1667, A 0.000, B 0.000, C 0.000 }
gfCNCPoint1[28026] = {X 98.8176, Y 47.3903, Z -2.1667, A 0.000, B 0.000, C 0.000 }
gfCNCPoint1[28027] = {X 98.3579, Y 46.5692, Z -2.1667, A 0.000, B 0.000, C 0.000 }
gfCNCPoint1[28028] = {X 94.8912, Y 38.0911, Z -2.1667, A 0.000, B 0.000, C 0.000 }
gfCNCPoint1[28029] = {X 94.8900, Y 38.2310, Z -2.1667, A 0.000, B 0.000, C 0.000 }
gfCNCPoint1[28030] = {X 94.8902, Y 41.0173, Z -2.1667, A 0.000, B 0.000, C 0.000 }
gfCNCPoint1[28031] = {X 95.4396, Y 41.5591, Z -2.1667, A 0.000, B 0.000, C 0.000 }
gfCNCPoint1[28032] = {X 95.8797, Y 42.1929, Z -2.1667, A 0.000, B 0.000, C 0.000 }
gfCNCPoint1[28033] = {X 96.1087, Y 42.6655, Z -2.1667, A 0.000, B 0.000, C 0.000 }
gfCNCPoint1[28034] = {X 96.2764, Y 43.1631, Z -2.1667, A 0.000, B 0.000, C 0.000 }
gfCNCPoint1[28035] = {X 96.3807, Y 43.6811, Z -2.1667, A 0.000, B 0.000, C 0.000 }
gfCNCPoint1[28036] = {X 96.4185, Y 44.2083, Z -2.1667, A 0.000, B 0.000, C 0.000 }
gfCNCPoint1[28037] = {X 96.4184, Y 45.0392, Z -2.1667, A 0.000, B 0.000, C 0.000 }
gfCNCPoint1[28038] = {X 96.3086, Y 45.9406, Z -2.1667, A 0.000, B 0.000, C 0.000 }
gfCNCPoint1[28039] = {X 96.0023, Y 46.7954, Z -2.1667, A 0.000, B 0.000, C 0.000 }
gfCNCPoint1[28040] = {X 95.5144, Y 47.5613, Z -2.1667, A 0.000, B 0.000, C 0.000 }
gfCNCPoint1[28041] = {X 94.8692, Y 48.2003, Z -2.1667, A 0.000, B 0.000, C 0.000 }
gfCNCPoint1[28042] = {X 94.0987, Y 48.6808, Z -2.1667, A 0.000, B 0.000, C 0.000 }
gfCNCPoint1[28043] = {X 93.2410, Y 48.9789, Z -2.1667, A 0.000, B 0.000, C 0.000 }
gfCNCPoint1[28044] = {X 92.3385, Y 49.0800, Z -2.1667, A 0.000, B 0.000, C 0.000 }
gfCNCPoint1[28045] = {X 85.8951, Y 49.0800, Z -2.1667, A 0.000, B 0.000, C 0.000 }
gfCNCPoint1[28046] = {X 84.9918, Y 48.9788, Z -2.1667, A 0.000, B 0.000, C 0.000 }
gfCNCPoint1[28047] = {X 84.1334, Y 48.6801, Z -2.1667, A 0.000, B 0.000, C 0.000 }
gfCNCPoint1[28048] = {X 83.3624, Y 48.1987, Z -2.1667, A 0.000, B 0.000, C 0.000 }
gfCNCPoint1[28049] = {X 82.7171, Y 47.5586, Z -2.1667, A 0.000, B 0.000, C 0.000 }
gfCNCPoint1[28050] = {X 82.2295, Y 46.7916, Z -2.1667, A 0.000, B 0.000, C 0.000 }
gfCNCPoint1[28051] = {X 81.9238, Y 45.9356, Z -2.1667, A 0.000, B 0.000, C 0.000 }
gfCNCPoint1[28052] = {X 81.8152, Y 45.0332, Z -2.1667, A 0.000, B 0.000, C 0.000 }
gfCNCPoint1[28053] = {X 81.8151, Y 44.2084, Z -2.1667, A 0.000, B 0.000, C 0.000 }
gfCNCPoint1[28054] = {X 81.9212, Y 43.3036, Z -2.1667, A 0.000, B 0.000, C 0.000 }
gfCNCPoint1[28055] = {X 82.2225, Y 42.4438, Z -2.1667, A 0.000, B 0.000, C 0.000 }
gfCNCPoint1[28056] = {X 82.7044, Y 41.6707, Z -2.1667, A 0.000, B 0.000, C 0.000 }
gfCNCPoint1[28057] = {X 83.3437, Y 41.0217, Z -2.1667, A 0.000, B 0.000, C 0.000 }
gfCNCPoint1[28058] = {X 83.3436, Y 28.5922, Z -2.1667, A 0.000, B 0.000, C 0.000 }
gfCNCPoint1[28059] = {X 79.3436, Y 28.5922, Z -2.1667, A 0.000, B 0.000, C 0.000 }
gfCNCPoint1[28060] = {X 83.4236, Y 28.5922, Z -2.1667, A 0.000, B 0.000, C 0.000 }
gfCNCPoint1[28061] = {X 83.4234, Y 16.1230, Z -2.1667, A 0.000, B 0.000, C 0.000 }
gfCNCPoint1[28062] = {X 82.7811, Y 15.4886, Z -2.1667, A 0.000, B 0.000, C 0.000 }
gfCNCPoint1[28063] = {X 82.2974, Y 14.7263, Z -2.1667, A 0.000, B 0.000, C 0.000 }
gfCNCPoint1[28064] = {X 81.9969, Y 13.8750, Z -2.1667, A 0.000, B 0.000, C 0.000 }
gfCNCPoint1[28065] = {X 81.8951, Y 12.9779, Z -2.1667, A 0.000, B 0.000, C 0.000 }
gfCNCPoint1[28066] = {X 81.8951, Y 12.1868, Z -2.1667, A 0.000, B 0.000, C 0.000 }
gfCNCPoint1[28067] = {X 81.9954, Y 11.2967, Z -2.1667, A 0.000, B 0.000, C 0.000 }
gfCNCPoint1[28068] = {X 82.2912, Y 10.4513, Z -2.1667, A 0.000, B 0.000, C 0.000 }
gfCNCPoint1[28069] = {X 82.7677, Y 9.6929, Z -2.1667, A 0.000, B 0.000, C 0.000 }
gfCNCPoint1[28070] = {X 83.4011, Y 9.0595, Z -2.1667, A 0.000, B 0.000, C 0.000 }
gfCNCPoint1[28071] = {X 84.1595, Y 8.5829, Z -2.1667, A 0.000, B 0.000, C 0.000 }
gfCNCPoint1[28072] = {X 85.0050, Y 8.2871, Z -2.1667, A 0.000, B 0.000, C 0.000 }
gfCNCPoint1[28073] = {X 85.8951, Y 8.1868, Z -2.1667, A 0.000, B 0.000, C 0.000 }
gfCNCPoint1[28074] = {X 94.0497, Y 8.1868, Z -2.1667, A 0.000, B 0.000, C 0.000 }
gfCNCPoint1[28075] = {X 94.9398, Y 8.2871, Z -2.1667, A 0.000, B 0.000, C 0.000 }
gfCNCPoint1[28076] = {X 95.7852, Y 8.5829, Z -2.1667, A 0.000, B 0.000, C 0.000 }
gfCNCPoint1[28077] = {X 96.5436, Y 9.0595, Z -2.1667, A 0.000, B 0.000, C 0.000 }
gfCNCPoint1[28078] = {X 97.1770, Y 9.6929, Z -2.1667, A 0.000, B 0.000, C 0.000 }
gfCNCPoint1[28079] = {X 97.6535, Y 10.4513, Z -2.1667, A 0.000, B 0.000, C 0.000 }
gfCNCPoint1[28080] = {X 97.9494, Y 11.2967, Z -2.1667, A 0.000, B 0.000, C 0.000 }
gfCNCPoint1[28081] = {X 98.0497, Y 12.1868, Z -2.1667, A 0.000, B 0.000, C 0.000 }
gfCNCPoint1[28082] = {X 98.0495, Y 13.0192, Z -2.1667, A 0.000, B 0.000, C 0.000 }
gfCNCPoint1[28083] = {X 97.9793, Y 13.7248, Z -2.1667, A 0.000, B 0.000, C 0.000 }
gfCNCPoint1[28084] = {X 97.7857, Y 14.4070, Z -2.1667, A 0.000, B 0.000, C 0.000 }
gfCNCPoint1[28085] = {X 97.4747, Y 15.0442, Z -2.1667, A 0.000, B 0.000, C 0.000 }
gfCNCPoint1[28086] = {X 97.4126, Y 15.1438, Z -2.1667, A 0.000, B 0.000, C 0.000 }
gfCNCPoint1[28087] = {X 97.3476, Y 15.2415, Z -2.1667, A 0.000, B 0.000, C 0.000 }
gfCNCPoint1[28088] = {X 97.4102, Y 15.3108, Z -2.1667, A 0.000, B 0.000, C 0.000 }
gfCNCPoint1[28089] = {X 97.9958, Y 16.7687, Z -2.1667, A 0.000, B 0.000, C 0.000 }
gfCNCPoint1[28090] = {X 101.6266, Y 25.7689, Z -2.1667, A 0.000, B 0.000, C 0.000 }
gfCNCPoint1[28091] = {X 101.8768, Y 26.3805, Z -2.1667, A 0.000, B 0.000, C 0.000 }
gfCNCPoint1[28092] = {X 102.1272, Y 25.7689, Z -2.1667, A 0.000, B 0.000, C 0.000 }
gfCNCPoint1[28093] = {X 106.3429, Y 15.2553, Z -2.1667, A 0.000, B 0.000, C 0.000 }
gfCNCPoint1[28094] = {X 106.3813, Y 15.1986, Z -2.1667, A 0.000, B 0.000, C 0.000 }
gfCNCPoint1[28095] = {X 106.3237, Y 15.1099, Z -2.1667, A 0.000, B 0.000, C 0.000 }
gfCNCPoint1[28096] = {X 106.2685, Y 15.0196, Z -2.1667, A 0.000, B 0.000, C 0.000 }
gfCNCPoint1[28097] = {X 105.9606, Y 14.3762, Z -2.1667, A 0.000, B 0.000, C 0.000 }
gfCNCPoint1[28098] = {X 105.7719, Y 13.6884, Z -2.1667, A 0.000, B 0.000, C 0.000 }
gfCNCPoint1[28099] = {X 105.7083, Y 12.9779, Z -2.1667, A 0.000, B 0.000, C 0.000 }
gfCNCPoint1[28100] = {X 105.7083, Y 12.1868, Z -2.1667, A 0.000, B 0.000, C 0.000 }
gfCNCPoint1[28101] = {X 105.8086, Y 11.2967, Z -2.1667, A 0.000, B 0.000, C 0.000 }
gfCNCPoint1[28102] = {X 106.1044, Y 10.4513, Z -2.1667, A 0.000, B 0.000, C 0.000 }
gfCNCPoint1[28103] = {X 106.5810, Y 9.6929, Z -2.1667, A 0.000, B 0.000, C 0.000 }
gfCNCPoint1[28104] = {X 107.2143, Y 9.0595, Z -2.1667, A 0.000, B 0.000, C 0.000 }
gfCNCPoint1[28105] = {X 107.9727, Y 8.5829, Z -2.1667, A 0.000, B 0.000, C 0.000 }
gfCNCPoint1[28106] = {X 108.8182, Y 8.2871, Z -2.1667, A 0.000, B 0.000, C 0.000 }
gfCNCPoint1[28107] = {X 109.7083, Y 8.1868, Z -2.1667, A 0.000, B 0.000, C 0.000 }
gfCNCPoint1[28108] = {X 117.7916, Y 8.1868, Z -2.1667, A 0.000, B 0.000, C 0.000 }
gfCNCPoint1[28109] = {X 118.6817, Y 8.2871, Z -2.1667, A 0.000, B 0.000, C 0.000 }
gfCNCPoint1[28110] = {X 119.5271, Y 8.5829, Z -2.1667, A 0.000, B 0.000, C 0.000 }
gfCNCPoint1[28111] = {X 120.2855, Y 9.0595, Z -2.1667, A 0.000, B 0.000, C 0.000 }
gfCNCPoint1[28112] = {X 120.9189, Y 9.6929, Z -2.1667, A 0.000, B 0.000, C 0.000 }
gfCNCPoint1[28113] = {X 121.3955, Y 10.4513, Z -2.1667, A 0.000, B 0.000, C 0.000 }
gfCNCPoint1[28114] = {X 121.6913, Y 11.2967, Z -2.1667, A 0.000, B 0.000, C 0.000 }
gfCNCPoint1[28115] = {X 121.7916, Y 12.1868, Z -2.1667, A 0.000, B 0.000, C 0.000 }
gfCNCPoint1[28116] = {X 121.7914, Y 13.0192, Z -2.1667, A 0.000, B 0.000, C 0.000 }
gfCNCPoint1[28117] = {X 121.6827, Y 13.9047, Z -2.1667, A 0.000, B 0.000, C 0.000 }
gfCNCPoint1[28118] = {X 121.3805, Y 14.7442, Z -2.1667, A 0.000, B 0.000, C 0.000 }
gfCNCPoint1[28119] = {X 120.8998, Y 15.4958, Z -2.1667, A 0.000, B 0.000, C 0.000 }
gfCNCPoint1[28120] = {X 120.2644, Y 16.1221, Z -2.1667, A 0.000, B 0.000, C 0.000 }
gfCNCPoint1[28121] = {X 120.2631, Y 41.0663, Z -2.1667, A 0.000, B 0.000, C 0.000 }
gfCNCPoint1[28122] = {X 120.4160, Y 41.1901, Z -2.1667, A 0.000, B 0.000, C 0.000 }
gfCNCPoint1[28123] = {X 120.9967, Y 41.8157, Z -2.1667, A 0.000, B 0.000, C 0.000 }
gfCNCPoint1[28124] = {X 121.4315, Y 42.5502, Z -2.1667, A 0.000, B 0.000, C 0.000 }
gfCNCPoint1[28125] = {X 121.7005, Y 43.3602, Z -2.1667, A 0.000, B 0.000, C 0.000 }
gfCNCPoint1[28126] = {X 121.7916, Y 44.2089, Z -2.1667, A 0.000, B 0.000, C 0.000 }
gfCNCPoint1[28127] = {X 121.7916, Y 45.0000, Z -2.1667, A 0.000, B 0.000, C 0.000 }
gfCNCPoint1[28128] = {X 121.6913, Y 45.8901, Z -2.1667, A 0.000, B 0.000, C 0.000 }
gfCNCPoint1[28129] = {X 121.3955, Y 46.7355, Z -2.1667, A 0.000, B 0.000, C 0.000 }
gfCNCPoint1[28130] = {X 120.9189, Y 47.4940, Z -2.1667, A 0.000, B 0.000, C 0.000 }
gfCNCPoint1[28131] = {X 120.2855, Y 48.1273, Z -2.1667, A 0.000, B 0.000, C 0.000 }
gfCNCPoint1[28132] = {X 119.5271, Y 48.6039, Z -2.1667, A 0.000, B 0.000, C 0.000 }
gfCNCPoint1[28133] = {X 118.6817, Y 48.8997, Z -2.1667, A 0.000, B 0.000, C 0.000 }
gfCNCPoint1[28134] = {X 117.7916, Y 49.0000, Z -2.1667, A 0.000, B 0.000, C 0.000 }
gfCNCPoint1[28135] = {X 111.9185, Y 49.0000, Z -2.1667, A 0.000, B 0.000, C 0.000 }
gfCNCPoint1[28136] = {X 111.0284, Y 48.8997, Z -2.1667, A 0.000, B 0.000, C 0.000 }
gfCNCPoint1[28137] = {X 110.1829, Y 48.6039, Z -2.1667, A 0.000, B 0.000, C 0.000 }
gfCNCPoint1[28138] = {X 109.4245, Y 48.1273, Z -2.1667, A 0.000, B 0.000, C 0.000 }
gfCNCPoint1[28139] = {X 108.7911, Y 47.4939, Z -2.1667, A 0.000, B 0.000, C 0.000 }
gfCNCPoint1[28140] = {X 108.3146, Y 46.7355, Z -2.1667, A 0.000, B 0.000, C 0.000 }
gfCNCPoint1[28141] = {X 108.0188, Y 45.8900, Z -2.1667, A 0.000, B 0.000, C 0.000 }
gfCNCPoint1[28142] = {X 107.9185, Y 45.0000, Z -2.1667, A 0.000, B 0.000, C 0.000 }
gfCNCPoint1[28143] = {X 107.9185, Y 44.1778, Z -2.1667, A 0.000, B 0.000, C 0.000 }
gfCNCPoint1[28144] = {X 107.9514, Y 43.6772, Z -2.1667, A 0.000, B 0.000, C 0.000 }
gfCNCPoint1[28145] = {X 108.0495, Y 43.1853, Z -2.1667, A 0.000, B 0.000, C 0.000 }
gfCNCPoint1[28146] = {X 108.2203, Y 42.6890, Z -2.1667, A 0.000, B 0.000, C 0.000 }
gfCNCPoint1[28147] = {X 108.4575, Y 42.2206, Z -2.1667, A 0.000, B 0.000, C 0.000 }
gfCNCPoint1[28148] = {X 108.9083, Y 41.5747, Z -2.1667, A 0.000, B 0.000, C 0.000 }
gfCNCPoint1[28149] = {X 109.4469, Y 40.9999, Z -2.1667, A 0.000, B 0.000, C 0.000 }
gfCNCPoint1[28150] = {X 109.4468, Y 38.9229, Z -2.1667, A 0.000, B 0.000, C 0.000 }
gfCNCPoint1[28151] = {X 108.9328, Y 38.9229, Z -2.1667, A 0.000, B 0.000, C 0.000 }
gfCNCPoint1[28152] = {X 105.8164, Y 46.5384, Z -2.1667, A 0.000, B 0.000, C 0.000 }
gfCNCPoint1[28153] = {X 105.3339, Y 47.3869, Z -2.1667, A 0.000, B 0.000, C 0.000 }
gfCNCPoint1[28154] = {X 104.6602, Y 48.0932, Z -2.1667, A 0.000, B 0.000, C 0.000 }
gfCNCPoint1[28155] = {X 103.8355, Y 48.6154, Z -2.1667, A 0.000, B 0.000, C 0.000 }
gfCNCPoint1[28156] = {X 102.9580, Y 48.9121, Z -2.1667, A 0.000, B 0.000, C 0.000 }
gfCNCPoint1[28157] = {X 102.0357, Y 48.9990, Z -2.1667, A 0.000, B 0.000, C 0.000 }
gfCNCPoint1[28158] = {X 101.1182, Y 48.8715, Z -2.1667, A 0.000, B 0.000, C 0.000 }
gfCNCPoint1[28159] = {X 100.2546, Y 48.5362, Z -2.1667, A 0.000, B 0.000, C 0.000 }
gfCNCPoint1[28160] = {X 99.4912, Y 48.0114, Z -2.1667, A 0.000, B 0.000, C 0.000 }
gfCNCPoint1[28161] = {X 98.8691, Y 47.3250, Z -2.1667, A 0.000, B 0.000, C 0.000 }
gfCNCPoint1[28162] = {X 98.4216, Y 46.5139, Z -2.1667, A 0.000, B 0.000, C 0.000 }
gfCNCPoint1[28163] = {X 94.8149, Y 37.6930, Z -2.1667, A 0.000, B 0.000, C 0.000 }
gfCNCPoint1[28164] = {X 94.8100, Y 38.2306, Z -2.1667, A 0.000, B 0.000, C 0.000 }
gfCNCPoint1[28165] = {X 94.8102, Y 41.0554, Z -2.1667, A 0.000, B 0.000, C 0.000 }
gfCNCPoint1[28166] = {X 95.3662, Y 41.5962, Z -2.1667, A 0.000, B 0.000, C 0.000 }
gfCNCPoint1[28167] = {X 95.8101, Y 42.2323, Z -2.1667, A 0.000, B 0.000, C 0.000 }
gfCNCPoint1[28168] = {X 96.0346, Y 42.6958, Z -2.1667, A 0.000, B 0.000, C 0.000 }
gfCNCPoint1[28169] = {X 96.1991, Y 43.1838, Z -2.1667, A 0.000, B 0.000, C 0.000 }
gfCNCPoint1[28170] = {X 96.3014, Y 43.6919, Z -2.1667, A 0.000, B 0.000, C 0.000 }
gfCNCPoint1[28171] = {X 96.3385, Y 44.2089, Z -2.1667, A 0.000, B 0.000, C 0.000 }
gfCNCPoint1[28172] = {X 96.3384, Y 45.0384, Z -2.1667, A 0.000, B 0.000, C 0.000 }
gfCNCPoint1[28173] = {X 96.2308, Y 45.9222, Z -2.1667, A 0.000, B 0.000, C 0.000 }
gfCNCPoint1[28174] = {X 95.9304, Y 46.7602, Z -2.1667, A 0.000, B 0.000, C 0.000 }
gfCNCPoint1[28175] = {X 95.4521, Y 47.5111, Z -2.1667, A 0.000, B 0.000, C 0.000 }
gfCNCPoint1[28176] = {X 94.8196, Y 48.1376, Z -2.1667, A 0.000, B 0.000, C 0.000 }
gfCNCPoint1[28177] = {X 94.0642, Y 48.6086, Z -2.1667, A 0.000, B 0.000, C 0.000 }
gfCNCPoint1[28178] = {X 93.2233, Y 48.9009, Z -2.1667, A 0.000, B 0.000, C 0.000 }
gfCNCPoint1[28179] = {X 92.3385, Y 49.0000, Z -2.1667, A 0.000, B 0.000, C 0.000 }
gfCNCPoint1[28180] = {X 85.8951, Y 49.0000, Z -2.1667, A 0.000, B 0.000, C 0.000 }
gfCNCPoint1[28181] = {X 85.0050, Y 48.8997, Z -2.1667, A 0.000, B 0.000, C 0.000 }
gfCNCPoint1[28182] = {X 84.1595, Y 48.6039, Z -2.1667, A 0.000, B 0.000, C 0.000 }
gfCNCPoint1[28183] = {X 83.4011, Y 48.1273, Z -2.1667, A 0.000, B 0.000, C 0.000 }
gfCNCPoint1[28184] = {X 82.7677, Y 47.4939, Z -2.1667, A 0.000, B 0.000, C 0.000 }
gfCNCPoint1[28185] = {X 82.2912, Y 46.7355, Z -2.1667, A 0.000, B 0.000, C 0.000 }
gfCNCPoint1[28186] = {X 81.9954, Y 45.8900, Z -2.1667, A 0.000, B 0.000, C 0.000 }
gfCNCPoint1[28187] = {X 81.8951, Y 45.0000, Z -2.1667, A 0.000, B 0.000, C 0.000 }
gfCNCPoint1[28188] = {X 81.8951, Y 44.2089, Z -2.1667, A 0.000, B 0.000, C 0.000 }
gfCNCPoint1[28189] = {X 82.0013, Y 43.3123, Z -2.1667, A 0.000, B 0.000, C 0.000 }
gfCNCPoint1[28190] = {X 82.3028, Y 42.4614, Z -2.1667, A 0.000, B 0.000, C 0.000 }
gfCNCPoint1[28191] = {X 82.7849, Y 41.6980, Z -2.1667, A 0.000, B 0.000, C 0.000 }
gfCNCPoint1[28192] = {X 83.4237, Y 41.0600, Z -2.1667, A 0.000, B 0.000, C 0.000 }
gfCNCPoint1[28193] = {X 83.4236, Y 28.5922, Z -2.1667, A 0.000, B 0.000, C 0.000 }
gfCNCPoint1[28194] = {X 79.3436, Y 28.5922, Z -2.1667, A 0.000, B 0.000, C 0.000 }
gfCNCPoint1[28195] = {X 79.3436, Y 28.5922, Z 0.8333, A 0.000, B 0.000, C 0.000 }
gfCNCPoint1[28196] = {X 79.3436, Y 28.5922, Z 11.0000, A 0.000, B 0.000, C 0.000 }
gfCNCPoint1[28197] = {X 136.1636, Y 30.3962, Z 11.0000, A 0.000, B 0.000, C 0.000 }
gfCNCPoint1[28198] = {X 136.1636, Y 30.3962, Z 0.8333, A 0.000, B 0.000, C 0.000 }
gfCNCPoint1[28199] = {X 136.1636, Y 30.3962, Z -2.1667, A 0.000, B 0.000, C 0.000 }
gfCNCPoint1[28200] = {X 140.2436, Y 30.3962, Z -2.1667, A 0.000, B 0.000, C 0.000 }
gfCNCPoint1[28201] = {X 140.2436, Y 19.8767, Z -2.1667, A 0.000, B 0.000, C 0.000 }
gfCNCPoint1[28202] = {X 137.4243, Y 19.8764, Z -2.1667, A 0.000, B 0.000, C 0.000 }
gfCNCPoint1[28203] = {X 136.8919, Y 20.5213, Z -2.1667, A 0.000, B 0.000, C 0.000 }
gfCNCPoint1[28204] = {X 136.2453, Y 21.0515, Z -2.1667, A 0.000, B 0.000, C 0.000 }
gfCNCPoint1[28205] = {X 135.5086, Y 21.4473, Z -2.1667, A 0.000, B 0.000, C 0.000 }
gfCNCPoint1[28206] = {X 134.7094, Y 21.6936, Z -2.1667, A 0.000, B 0.000, C 0.000 }
gfCNCPoint1[28207] = {X 133.8778, Y 21.7814, Z -2.1667, A 0.000, B 0.000, C 0.000 }
gfCNCPoint1[28208] = {X 133.2006, Y 21.7815, Z -2.1667, A 0.000, B 0.000, C 0.000 }
gfCNCPoint1[28209] = {X 132.2394, Y 21.6732, Z -2.1667, A 0.000, B 0.000, C 0.000 }
gfCNCPoint1[28210] = {X 131.3263, Y 21.3537, Z -2.1667, A 0.000, B 0.000, C 0.000 }
gfCNCPoint1[28211] = {X 130.5072, Y 20.8390, Z -2.1667, A 0.000, B 0.000, C 0.000 }
gfCNCPoint1[28212] = {X 129.8231, Y 20.1550, Z -2.1667, A 0.000, B 0.000, C 0.000 }
gfCNCPoint1[28213] = {X 129.3085, Y 19.3359, Z -2.1667, A 0.000, B 0.000, C 0.000 }
gfCNCPoint1[28214] = {X 128.9890, Y 18.4228, Z -2.1667, A 0.000, B 0.000, C 0.000 }
gfCNCPoint1[28215] = {X 128.8806, Y 17.4615, Z -2.1667, A 0.000, B 0.000, C 0.000 }
gfCNCPoint1[28216] = {X 128.8806, Y 10.4835, Z -2.1667, A 0.000, B 0.000, C 0.000 }
gfCNCPoint1[28217] = {X 128.9874, Y 9.5289, Z -2.1667, A 0.000, B 0.000, C 0.000 }
gfCNCPoint1[28218] = {X 129.3026, Y 8.6214, Z -2.1667, A 0.000, B 0.000, C 0.000 }
gfCNCPoint1[28219] = {X 129.8104, Y 7.8061, Z -2.1667, A 0.000, B 0.000, C 0.000 }
gfCNCPoint1[28220] = {X 130.4859, Y 7.1231, Z -2.1667, A 0.000, B 0.000, C 0.000 }
gfCNCPoint1[28221] = {X 131.2956, Y 6.6063, Z -2.1667, A 0.000, B 0.000, C 0.000 }
gfCNCPoint1[28222] = {X 132.1995, Y 6.2811, Z -2.1667, A 0.000, B 0.000, C 0.000 }
gfCNCPoint1[28223] = {X 133.1529, Y 6.1638, Z -2.1667, A 0.000, B 0.000, C 0.000 }
gfCNCPoint1[28224] = {X 133.8866, Y 6.1637, Z -2.1667, A 0.000, B 0.000, C 0.000 }
gfCNCPoint1[28225] = {X 134.7113, Y 6.2518, Z -2.1667, A 0.000, B 0.000, C 0.000 }
gfCNCPoint1[28226] = {X 135.5040, Y 6.4959, Z -2.1667, A 0.000, B 0.000, C 0.000 }
gfCNCPoint1[28227] = {X 136.2354, Y 6.8869, Z -2.1667, A 0.000, B 0.000, C 0.000 }
gfCNCPoint1[28228] = {X 136.8786, Y 7.4105, Z -2.1667, A 0.000, B 0.000, C 0.000 }
gfCNCPoint1[28229] = {X 137.4099, Y 8.0474, Z -2.1667, A 0.000, B 0.000, C 0.000 }
gfCNCPoint1[28230] = {X 155.1121, Y 8.0485, Z -2.1667, A 0.000, B 0.000, C 0.000 }
gfCNCPoint1[28231] = {X 155.6441, Y 7.4105, Z -2.1667, A 0.000, B 0.000, C 0.000 }
gfCNCPoint1[28232] = {X 156.2884, Y 6.8862, Z -2.1667, A 0.000, B 0.000, C 0.000 }
gfCNCPoint1[28233] = {X 157.0211, Y 6.4949, Z -2.1667, A 0.000, B 0.000, C 0.000 }
gfCNCPoint1[28234] = {X 157.8152, Y 6.2511, Z -2.1667, A 0.000, B 0.000, C 0.000 }
gfCNCPoint1[28235] = {X 158.6412, Y 6.1637, Z -2.1667, A 0.000, B 0.000, C 0.000 }
gfCNCPoint1[28236] = {X 159.3781, Y 6.1639, Z -2.1667, A 0.000, B 0.000, C 0.000 }
gfCNCPoint1[28237] = {X 160.3301, Y 6.2828, Z -2.1667, A 0.000, B 0.000, C 0.000 }
gfCNCPoint1[28238] = {X 161.2324, Y 6.6088, Z -2.1667, A 0.000, B 0.000, C 0.000 }
gfCNCPoint1[28239] = {X 162.0405, Y 7.1260, Z -2.1667, A 0.000, B 0.000, C 0.000 }
gfCNCPoint1[28240] = {X 162.7145, Y 7.8088, Z -2.1667, A 0.000, B 0.000, C 0.000 }
gfCNCPoint1[28241] = {X 163.2212, Y 8.6236, Z -2.1667, A 0.000, B 0.000, C 0.000 }
gfCNCPoint1[28242] = {X 163.5355, Y 9.5300, Z -2.1667, A 0.000, B 0.000, C 0.000 }
gfCNCPoint1[28243] = {X 163.6421, Y 10.4835, Z -2.1667, A 0.000, B 0.000, C 0.000 }
gfCNCPoint1[28244] = {X 163.6421, Y 17.4615, Z -2.1667, A 0.000, B 0.000, C 0.000 }
gfCNCPoint1[28245] = {X 163.5355, Y 18.4152, Z -2.1667, A 0.000, B 0.000, C 0.000 }
gfCNCPoint1[28246] = {X 163.2211, Y 19.3218, Z -2.1667, A 0.000, B 0.000, C 0.000 }
gfCNCPoint1[28247] = {X 162.7142, Y 20.1366, Z -2.1667, A 0.000, B 0.000, C 0.000 }
gfCNCPoint1[28248] = {X 162.0400, Y 20.8194, Z -2.1667, A 0.000, B 0.000, C 0.000 }
gfCNCPoint1[28249] = {X 161.2318, Y 21.3365, Z -2.1667, A 0.000, B 0.000, C 0.000 }
gfCNCPoint1[28250] = {X 160.3292, Y 21.6625, Z -2.1667, A 0.000, B 0.000, C 0.000 }
gfCNCPoint1[28251] = {X 159.3770, Y 21.7812, Z -2.1667, A 0.000, B 0.000, C 0.000 }
gfCNCPoint1[28252] = {X 158.6790, Y 21.7815, Z -2.1667, A 0.000, B 0.000, C 0.000 }
gfCNCPoint1[28253] = {X 157.8407, Y 21.6960, Z -2.1667, A 0.000, B 0.000, C 0.000 }
gfCNCPoint1[28254] = {X 157.0346, Y 21.4507, Z -2.1667, A 0.000, B 0.000, C 0.000 }
gfCNCPoint1[28255] = {X 156.2907, Y 21.0549, Z -2.1667, A 0.000, B 0.000, C 0.000 }
gfCNCPoint1[28256] = {X 155.6368, Y 20.5234, Z -2.1667, A 0.000, B 0.000, C 0.000 }
gfCNCPoint1[28257] = {X 155.0975, Y 19.8760, Z -2.1667, A 0.000, B 0.000, C 0.000 }
gfCNCPoint1[28258] = {X 152.2758, Y 19.8774, Z -2.1667, A 0.000, B 0.000, C 0.000 }
gfCNCPoint1[28259] = {X 152.2741, Y 40.8742, Z -2.1667, A 0.000, B 0.000, C 0.000 }
gfCNCPoint1[28260] = {X 152.7410, Y 41.3767, Z -2.1667, A 0.000, B 0.000, C 0.000 }
gfCNCPoint1[28261] = {X 152.8350, Y 41.4890, Z -2.1667, A 0.000, B 0.000, C 0.000 }
gfCNCPoint1[28262] = {X 153.3603, Y 42.3142, Z -2.1667, A 0.000, B 0.000, C 0.000 }
gfCNCPoint1[28263] = {X 153.6885, Y 43.2358, Z -2.1667, A 0.000, B 0.000, C 0.000 }
gfCNCPoint1[28264] = {X 153.8031, Y 44.2073, Z -2.1667, A 0.000, B 0.000, C 0.000 }
gfCNCPoint1[28265] = {X 153.8029, Y 45.0415, Z -2.1667, A 0.000, B 0.000, C 0.000 }
gfCNCPoint1[28266] = {X 153.6867, Y 45.9960, Z -2.1667, A 0.000, B 0.000, C 0.000 }
gfCNCPoint1[28267] = {X 153.3623, Y 46.9011, Z -2.1667, A 0.000, B 0.000, C 0.000 }
gfCNCPoint1[28268] = {X 152.8458, Y 47.7120, Z -2.1667, A 0.000, B 0.000, C 0.000 }
gfCNCPoint1[28269] = {X 152.1626, Y 48.3886, Z -2.1667, A 0.000, B 0.000, C 0.000 }
gfCNCPoint1[28270] = {X 151.3468, Y 48.8973, Z -2.1667, A 0.000, B 0.000, C 0.000 }
gfCNCPoint1[28271] = {X 150.4386, Y 49.2130, Z -2.1667, A 0.000, B 0.000, C 0.000 }
gfCNCPoint1[28272] = {X 149.4831, Y 49.3200, Z -2.1667, A 0.000, B 0.000, C 0.000 }
gfCNCPoint1[28273] = {X 143.0396, Y 49.3200, Z -2.1667, A 0.000, B 0.000, C 0.000 }
gfCNCPoint1[28274] = {X 142.0831, Y 49.2128, Z -2.1667, A 0.000, B 0.000, C 0.000 }
gfCNCPoint1[28275] = {X 141.1741, Y 48.8964, Z -2.1667, A 0.000, B 0.000, C 0.000 }
gfCNCPoint1[28276] = {X 140.3576, Y 48.3866, Z -2.1667, A 0.000, B 0.000, C 0.000 }
gfCNCPoint1[28277] = {X 139.6743, Y 47.7087, Z -2.1667, A 0.000, B 0.000, C 0.000 }
gfCNCPoint1[28278] = {X 139.1581, Y 46.8964, Z -2.1667, A 0.000, B 0.000, C 0.000 }
gfCNCPoint1[28279] = {X 138.8346, Y 45.9899, Z -2.1667, A 0.000, B 0.000, C 0.000 }
gfCNCPoint1[28280] = {X 138.7198, Y 45.0342, Z -2.1667, A 0.000, B 0.000, C 0.000 }
gfCNCPoint1[28281] = {X 138.7200, Y 44.1494, Z -2.1667, A 0.000, B 0.000, C 0.000 }
gfCNCPoint1[28282] = {X 138.8305, Y 43.2364, Z -2.1667, A 0.000, B 0.000, C 0.000 }
gfCNCPoint1[28283] = {X 139.1317, Y 42.3675, Z -2.1667, A 0.000, B 0.000, C 0.000 }
gfCNCPoint1[28284] = {X 139.6099, Y 41.5821, Z -2.1667, A 0.000, B 0.000, C 0.000 }
gfCNCPoint1[28285] = {X 140.2436, Y 40.9157, Z -2.1667, A 0.000, B 0.000, C 0.000 }
gfCNCPoint1[28286] = {X 140.2436, Y 30.3962, Z -2.1667, A 0.000, B 0.000, C 0.000 }
gfCNCPoint1[28287] = {X 136.2436, Y 30.3962, Z -2.1667, A 0.000, B 0.000, C 0.000 }
gfCNCPoint1[28288] = {X 140.3236, Y 30.3962, Z -2.1667, A 0.000, B 0.000, C 0.000 }
gfCNCPoint1[28289] = {X 140.3236, Y 19.7968, Z -2.1667, A 0.000, B 0.000, C 0.000 }
gfCNCPoint1[28290] = {X 137.3800, Y 19.7959, Z -2.1667, A 0.000, B 0.000, C 0.000 }
gfCNCPoint1[28291] = {X 137.3571, Y 19.8330, Z -2.1667, A 0.000, B 0.000, C 0.000 }
gfCNCPoint1[28292] = {X 136.8346, Y 20.4655, Z -2.1667, A 0.000, B 0.000, C 0.000 }
gfCNCPoint1[28293] = {X 136.2000, Y 20.9856, Z -2.1667, A 0.000, B 0.000, C 0.000 }
gfCNCPoint1[28294] = {X 135.4771, Y 21.3737, Z -2.1667, A 0.000, B 0.000, C 0.000 }
gfCNCPoint1[28295] = {X 134.6931, Y 21.6153, Z -2.1667, A 0.000, B 0.000, C 0.000 }
gfCNCPoint1[28296] = {X 133.8772, Y 21.7014, Z -2.1667, A 0.000, B 0.000, C 0.000 }
gfCNCPoint1[28297] = {X 133.2006, Y 21.7015, Z -2.1667, A 0.000, B 0.000, C 0.000 }
gfCNCPoint1[28298] = {X 132.2572, Y 21.5952, Z -2.1667, A 0.000, B 0.000, C 0.000 }
gfCNCPoint1[28299] = {X 131.3610, Y 21.2816, Z -2.1667, A 0.000, B 0.000, C 0.000 }
gfCNCPoint1[28300] = {X 130.5570, Y 20.7765, Z -2.1667, A 0.000, B 0.000, C 0.000 }
gfCNCPoint1[28301] = {X 129.8857, Y 20.1051, Z -2.1667, A 0.000, B 0.000, C 0.000 }
gfCNCPoint1[28302] = {X 129.3805, Y 19.3012, Z -2.1667, A 0.000, B 0.000, C 0.000 }
gfCNCPoint1[28303] = {X 129.0669, Y 18.4050, Z -2.1667, A 0.000, B 0.000, C 0.000 }
gfCNCPoint1[28304] = {X 128.9606, Y 17.4615, Z -2.1667, A 0.000, B 0.000, C 0.000 }
gfCNCPoint1[28305] = {X 128.9606, Y 10.4835, Z -2.1667, A 0.000, B 0.000, C 0.000 }
gfCNCPoint1[28306] = {X 129.0655, Y 9.5466, Z -2.1667, A 0.000, B 0.000, C 0.000 }
gfCNCPoint1[28307] = {X 129.3747, Y 8.6559, Z -2.1667, A 0.000, B 0.000, C 0.000 }
gfCNCPoint1[28308] = {X 129.8732, Y 7.8557, Z -2.1667, A 0.000, B 0.000, C 0.000 }
gfCNCPoint1[28309] = {X 130.5362, Y 7.1853, Z -2.1667, A 0.000, B 0.000, C 0.000 }
gfCNCPoint1[28310] = {X 131.3309, Y 6.6781, Z -2.1667, A 0.000, B 0.000, C 0.000 }
gfCNCPoint1[28311] = {X 132.2180, Y 6.3589, Z -2.1667, A 0.000, B 0.000, C 0.000 }
gfCNCPoint1[28312] = {X 133.1538, Y 6.2438, Z -2.1667, A 0.000, B 0.000, C 0.000 }
gfCNCPoint1[28313] = {X 133.8858, Y 6.2437, Z -2.1667, A 0.000, B 0.000, C 0.000 }
gfCNCPoint1[28314] = {X 134.7034, Y 6.3319, Z -2.1667, A 0.000, B 0.000, C 0.000 }
gfCNCPoint1[28315] = {X 135.4887, Y 6.5762, Z -2.1667, A 0.000, B 0.000, C 0.000 }
gfCNCPoint1[28316] = {X 136.2120, Y 6.9676, Z -2.1667, A 0.000, B 0.000, C 0.000 }
gfCNCPoint1[28317] = {X 136.8462, Y 7.4912, Z -2.1667, A 0.000, B 0.000, C 0.000 }
gfCNCPoint1[28318] = {X 137.3674, Y 8.1274, Z -2.1667, A 0.000, B 0.000, C 0.000 }
gfCNCPoint1[28319] = {X 155.1546, Y 8.1285, Z -2.1667, A 0.000, B 0.000, C 0.000 }
gfCNCPoint1[28320] = {X 155.6765, Y 7.4912, Z -2.1667, A 0.000, B 0.000, C 0.000 }
gfCNCPoint1[28321] = {X 156.3117, Y 6.9669, Z -2.1667, A 0.000, B 0.000, C 0.000 }
gfCNCPoint1[28322] = {X 157.0363, Y 6.5753, Z -2.1667, A 0.000, B 0.000, C 0.000 }
gfCNCPoint1[28323] = {X 157.8229, Y 6.3311, Z -2.1667, A 0.000, B 0.000, C 0.000 }
gfCNCPoint1[28324] = {X 158.6420, Y 6.2437, Z -2.1667, A 0.000, B 0.000, C 0.000 }
gfCNCPoint1[28325] = {X 159.3770, Y 6.2439, Z -2.1667, A 0.000, B 0.000, C 0.000 }
gfCNCPoint1[28326] = {X 160.3114, Y 6.3606, Z -2.1667, A 0.000, B 0.000, C 0.000 }
gfCNCPoint1[28327] = {X 161.1970, Y 6.6806, Z -2.1667, A 0.000, B 0.000, C 0.000 }
gfCNCPoint1[28328] = {X 161.9902, Y 7.1882, Z -2.1667, A 0.000, B 0.000, C 0.000 }
gfCNCPoint1[28329] = {X 162.6517, Y 7.8584, Z -2.1667, A 0.000, B 0.000, C 0.000 }
gfCNCPoint1[28330] = {X 163.1490, Y 8.6580, Z -2.1667, A 0.000, B 0.000, C 0.000 }
gfCNCPoint1[28331] = {X 163.4575, Y 9.5477, Z -2.1667, A 0.000, B 0.000, C 0.000 }
gfCNCPoint1[28332] = {X 163.5621, Y 10.4835, Z -2.1667, A 0.000, B 0.000, C 0.000 }
gfCNCPoint1[28333] = {X 163.5621, Y 17.4615, Z -2.1667, A 0.000, B 0.000, C 0.000 }
gfCNCPoint1[28334] = {X 163.4575, Y 18.3975, Z -2.1667, A 0.000, B 0.000, C 0.000 }
gfCNCPoint1[28335] = {X 163.1489, Y 19.2873, Z -2.1667, A 0.000, B 0.000, C 0.000 }
gfCNCPoint1[28336] = {X 162.6514, Y 20.0870, Z -2.1667, A 0.000, B 0.000, C 0.000 }
gfCNCPoint1[28337] = {X 161.9897, Y 20.7572, Z -2.1667, A 0.000, B 0.000, C 0.000 }
gfCNCPoint1[28338] = {X 161.1964, Y 21.2648, Z -2.1667, A 0.000, B 0.000, C 0.000 }
gfCNCPoint1[28339] = {X 160.3106, Y 21.5847, Z -2.1667, A 0.000, B 0.000, C 0.000 }
gfCNCPoint1[28340] = {X 159.3760, Y 21.7012, Z -2.1667, A 0.000, B 0.000, C 0.000 }
gfCNCPoint1[28341] = {X 158.6794, Y 21.7015, Z -2.1667, A 0.000, B 0.000, C 0.000 }
gfCNCPoint1[28342] = {X 157.8482, Y 21.6159, Z -2.1667, A 0.000, B 0.000, C 0.000 }
gfCNCPoint1[28343] = {X 157.0496, Y 21.3703, Z -2.1667, A 0.000, B 0.000, C 0.000 }
gfCNCPoint1[28344] = {X 156.3138, Y 20.9742, Z -2.1667, A 0.000, B 0.000, C 0.000 }
gfCNCPoint1[28345] = {X 155.6691, Y 20.4426, Z -2.1667, A 0.000, B 0.000, C 0.000 }
gfCNCPoint1[28346] = {X 155.1400, Y 19.7959, Z -2.1667, A 0.000, B 0.000, C 0.000 }
gfCNCPoint1[28347] = {X 152.1958, Y 19.7974, Z -2.1667, A 0.000, B 0.000, C 0.000 }
gfCNCPoint1[28348] = {X 152.1941, Y 40.9056, Z -2.1667, A 0.000, B 0.000, C 0.000 }
gfCNCPoint1[28349] = {X 152.6810, Y 41.4297, Z -2.1667, A 0.000, B 0.000, C 0.000 }
gfCNCPoint1[28350] = {X 152.7732, Y 41.5398, Z -2.1667, A 0.000, B 0.000, C 0.000 }
gfCNCPoint1[28351] = {X 153.2887, Y 42.3498, Z -2.1667, A 0.000, B 0.000, C 0.000 }
gfCNCPoint1[28352] = {X 153.6107, Y 43.2542, Z -2.1667, A 0.000, B 0.000, C 0.000 }
gfCNCPoint1[28353] = {X 153.7231, Y 44.2077, Z -2.1667, A 0.000, B 0.000, C 0.000 }
gfCNCPoint1[28354] = {X 153.7229, Y 45.0408, Z -2.1667, A 0.000, B 0.000, C 0.000 }
gfCNCPoint1[28355] = {X 153.6089, Y 45.9775, Z -2.1667, A 0.000, B 0.000, C 0.000 }
gfCNCPoint1[28356] = {X 153.2905, Y 46.8659, Z -2.1667, A 0.000, B 0.000, C 0.000 }
gfCNCPoint1[28357] = {X 152.7835, Y 47.6618, Z -2.1667, A 0.000, B 0.000, C 0.000 }
gfCNCPoint1[28358] = {X 152.1130, Y 48.3258, Z -2.1667, A 0.000, B 0.000, C 0.000 }
gfCNCPoint1[28359] = {X 151.3123, Y 48.8251, Z -2.1667, A 0.000, B 0.000, C 0.000 }
gfCNCPoint1[28360] = {X 150.4209, Y 49.1350, Z -2.1667, A 0.000, B 0.000, C 0.000 }
gfCNCPoint1[28361] = {X 149.4831, Y 49.2400, Z -2.1667, A 0.000, B 0.000, C 0.000 }
gfCNCPoint1[28362] = {X 143.0396, Y 49.2400, Z -2.1667, A 0.000, B 0.000, C 0.000 }
gfCNCPoint1[28363] = {X 142.1008, Y 49.1348, Z -2.1667, A 0.000, B 0.000, C 0.000 }
gfCNCPoint1[28364] = {X 141.2086, Y 48.8243, Z -2.1667, A 0.000, B 0.000, C 0.000 }
gfCNCPoint1[28365] = {X 140.4073, Y 48.3239, Z -2.1667, A 0.000, B 0.000, C 0.000 }
gfCNCPoint1[28366] = {X 139.7367, Y 47.6586, Z -2.1667, A 0.000, B 0.000, C 0.000 }
gfCNCPoint1[28367] = {X 139.2300, Y 46.8612, Z -2.1667, A 0.000, B 0.000, C 0.000 }
gfCNCPoint1[28368] = {X 138.9124, Y 45.9715, Z -2.1667, A 0.000, B 0.000, C 0.000 }
gfCNCPoint1[28369] = {X 138.7998, Y 45.0336, Z -2.1667, A 0.000, B 0.000, C 0.000 }
gfCNCPoint1[28370] = {X 138.8000, Y 44.1505, Z -2.1667, A 0.000, B 0.000, C 0.000 }
gfCNCPoint1[28371] = {X 138.9105, Y 43.2454, Z -2.1667, A 0.000, B 0.000, C 0.000 }
gfCNCPoint1[28372] = {X 139.2119, Y 42.3850, Z -2.1667, A 0.000, B 0.000, C 0.000 }
gfCNCPoint1[28373] = {X 139.6903, Y 41.6088, Z -2.1667, A 0.000, B 0.000, C 0.000 }
gfCNCPoint1[28374] = {X 140.3236, Y 40.9529, Z -2.1667, A 0.000, B 0.000, C 0.000 }
gfCNCPoint1[28375] = {X 140.3236, Y 30.3962, Z -2.1667, A 0.000, B 0.000, C 0.000 }
gfCNCPoint1[28376] = {X 136.3236, Y 30.3962, Z -2.1667, A 0.000, B 0.000, C 0.000 }
gfCNCPoint1[28377] = {X 140.4036, Y 30.3962, Z -2.1667, A 0.000, B 0.000, C 0.000 }
gfCNCPoint1[28378] = {X 140.4036, Y 19.7168, Z -2.1667, A 0.000, B 0.000, C 0.000 }
gfCNCPoint1[28379] = {X 137.3354, Y 19.7159, Z -2.1667, A 0.000, B 0.000, C 0.000 }
gfCNCPoint1[28380] = {X 137.2899, Y 19.7896, Z -2.1667, A 0.000, B 0.000, C 0.000 }
gfCNCPoint1[28381] = {X 136.7772, Y 20.4098, Z -2.1667, A 0.000, B 0.000, C 0.000 }
gfCNCPoint1[28382] = {X 136.1547, Y 20.9196, Z -2.1667, A 0.000, B 0.000, C 0.000 }
gfCNCPoint1[28383] = {X 135.4457, Y 21.3001, Z -2.1667, A 0.000, B 0.000, C 0.000 }
gfCNCPoint1[28384] = {X 134.6767, Y 21.5370, Z -2.1667, A 0.000, B 0.000, C 0.000 }
gfCNCPoint1[28385] = {X 133.8765, Y 21.6214, Z -2.1667, A 0.000, B 0.000, C 0.000 }
gfCNCPoint1[28386] = {X 133.2006, Y 21.6215, Z -2.1667, A 0.000, B 0.000, C 0.000 }
gfCNCPoint1[28387] = {X 132.2750, Y 21.5172, Z -2.1667, A 0.000, B 0.000, C 0.000 }
gfCNCPoint1[28388] = {X 131.3957, Y 21.2096, Z -2.1667, A 0.000, B 0.000, C 0.000 }
gfCNCPoint1[28389] = {X 130.6069, Y 20.7140, Z -2.1667, A 0.000, B 0.000, C 0.000 }
gfCNCPoint1[28390] = {X 129.9482, Y 20.0553, Z -2.1667, A 0.000, B 0.000, C 0.000 }
gfCNCPoint1[28391] = {X 129.4526, Y 19.2665, Z -2.1667, A 0.000, B 0.000, C 0.000 }
gfCNCPoint1[28392] = {X 129.1449, Y 18.3872, Z -2.1667, A 0.000, B 0.000, C 0.000 }
gfCNCPoint1[28393] = {X 129.0406, Y 17.4615, Z -2.1667, A 0.000, B 0.000, C 0.000 }
gfCNCPoint1[28394] = {X 129.0406, Y 10.4835, Z -2.1667, A 0.000, B 0.000, C 0.000 }
gfCNCPoint1[28395] = {X 129.1435, Y 9.5642, Z -2.1667, A 0.000, B 0.000, C 0.000 }
gfCNCPoint1[28396] = {X 129.4469, Y 8.6904, Z -2.1667, A 0.000, B 0.000, C 0.000 }
gfCNCPoint1[28397] = {X 129.9360, Y 7.9052, Z -2.1667, A 0.000, B 0.000, C 0.000 }
gfCNCPoint1[28398] = {X 130.5864, Y 7.2475, Z -2.1667, A 0.000, B 0.000, C 0.000 }
gfCNCPoint1[28399] = {X 131.3662, Y 6.7499, Z -2.1667, A 0.000, B 0.000, C 0.000 }
gfCNCPoint1[28400] = {X 132.2366, Y 6.4368, Z -2.1667, A 0.000, B 0.000, C 0.000 }
gfCNCPoint1[28401] = {X 133.1547, Y 6.3238, Z -2.1667, A 0.000, B 0.000, C 0.000 }
gfCNCPoint1[28402] = {X 133.8850, Y 6.3237, Z -2.1667, A 0.000, B 0.000, C 0.000 }
gfCNCPoint1[28403] = {X 134.6955, Y 6.4120, Z -2.1667, A 0.000, B 0.000, C 0.000 }
gfCNCPoint1[28404] = {X 135.4733, Y 6.6566, Z -2.1667, A 0.000, B 0.000, C 0.000 }
gfCNCPoint1[28405] = {X 136.1885, Y 7.0482, Z -2.1667, A 0.000, B 0.000, C 0.000 }
gfCNCPoint1[28406] = {X 136.8135, Y 7.5719, Z -2.1667, A 0.000, B 0.000, C 0.000 }
gfCNCPoint1[28407] = {X 137.3244, Y 8.2074, Z -2.1667, A 0.000, B 0.000, C 0.000 }
gfCNCPoint1[28408] = {X 155.1976, Y 8.2085, Z -2.1667, A 0.000, B 0.000, C 0.000 }
gfCNCPoint1[28409] = {X 155.7092, Y 7.5719, Z -2.1667, A 0.000, B 0.000, C 0.000 }
gfCNCPoint1[28410] = {X 156.3352, Y 7.0476, Z -2.1667, A 0.000, B 0.000, C 0.000 }
gfCNCPoint1[28411] = {X 157.0516, Y 6.6556, Z -2.1667, A 0.000, B 0.000, C 0.000 }
gfCNCPoint1[28412] = {X 157.8308, Y 6.4112, Z -2.1667, A 0.000, B 0.000, C 0.000 }
gfCNCPoint1[28413] = {X 158.6427, Y 6.3237, Z -2.1667, A 0.000, B 0.000, C 0.000 }
gfCNCPoint1[28414] = {X 159.3760, Y 6.3239, Z -2.1667, A 0.000, B 0.000, C 0.000 }
gfCNCPoint1[28415] = {X 160.2928, Y 6.4383, Z -2.1667, A 0.000, B 0.000, C 0.000 }
gfCNCPoint1[28416] = {X 161.1617, Y 6.7524, Z -2.1667, A 0.000, B 0.000, C 0.000 }
gfCNCPoint1[28417] = {X 161.9398, Y 7.2504, Z -2.1667, A 0.000, B 0.000, C 0.000 }
gfCNCPoint1[28418] = {X 162.5889, Y 7.9079, Z -2.1667, A 0.000, B 0.000, C 0.000 }
gfCNCPoint1[28419] = {X 163.0768, Y 8.6925, Z -2.1667, A 0.000, B 0.000, C 0.000 }
gfCNCPoint1[28420] = {X 163.3795, Y 9.5653, Z -2.1667, A 0.000, B 0.000, C 0.000 }
gfCNCPoint1[28421] = {X 163.4821, Y 10.4835, Z -2.1667, A 0.000, B 0.000, C 0.000 }
gfCNCPoint1[28422] = {X 163.4821, Y 17.4615, Z -2.1667, A 0.000, B 0.000, C 0.000 }
gfCNCPoint1[28423] = {X 163.3795, Y 18.3798, Z -2.1667, A 0.000, B 0.000, C 0.000 }
gfCNCPoint1[28424] = {X 163.0767, Y 19.2527, Z -2.1667, A 0.000, B 0.000, C 0.000 }
gfCNCPoint1[28425] = {X 162.5887, Y 20.0373, Z -2.1667, A 0.000, B 0.000, C 0.000 }
gfCNCPoint1[28426] = {X 161.9396, Y 20.6948, Z -2.1667, A 0.000, B 0.000, C 0.000 }
gfCNCPoint1[28427] = {X 161.1613, Y 21.1929, Z -2.1667, A 0.000, B 0.000, C 0.000 }
gfCNCPoint1[28428] = {X 160.2923, Y 21.5068, Z -2.1667, A 0.000, B 0.000, C 0.000 }
gfCNCPoint1[28429] = {X 159.3755, Y 21.6212, Z -2.1667, A 0.000, B 0.000, C 0.000 }
gfCNCPoint1[28430] = {X 158.6798, Y 21.6215, Z -2.1667, A 0.000, B 0.000, C 0.000 }
gfCNCPoint1[28431] = {X 157.8558, Y 21.5358, Z -2.1667, A 0.000, B 0.000, C 0.000 }
gfCNCPoint1[28432] = {X 157.0647, Y 21.2899, Z -2.1667, A 0.000, B 0.000, C 0.000 }
gfCNCPoint1[28433] = {X 156.3372, Y 20.8934, Z -2.1667, A 0.000, B 0.000, C 0.000 }
gfCNCPoint1[28434] = {X 155.7018, Y 20.3619, Z -2.1667, A 0.000, B 0.000, C 0.000 }
gfCNCPoint1[28435] = {X 155.1831, Y 19.7159, Z -2.1667, A 0.000, B 0.000, C 0.000 }
gfCNCPoint1[28436] = {X 152.1158, Y 19.7175, Z -2.1667, A 0.000, B 0.000, C 0.000 }
gfCNCPoint1[28437] = {X 152.1141, Y 40.9370, Z -2.1667, A 0.000, B 0.000, C 0.000 }
gfCNCPoint1[28438] = {X 152.6209, Y 41.4826, Z -2.1667, A 0.000, B 0.000, C 0.000 }
gfCNCPoint1[28439] = {X 152.7114, Y 41.5906, Z -2.1667, A 0.000, B 0.000, C 0.000 }
gfCNCPoint1[28440] = {X 153.2170, Y 42.3853, Z -2.1667, A 0.000, B 0.000, C 0.000 }
gfCNCPoint1[28441] = {X 153.5329, Y 43.2727, Z -2.1667, A 0.000, B 0.000, C 0.000 }
gfCNCPoint1[28442] = {X 153.6431, Y 44.2081, Z -2.1667, A 0.000, B 0.000, C 0.000 }
gfCNCPoint1[28443] = {X 153.6429, Y 45.0400, Z -2.1667, A 0.000, B 0.000, C 0.000 }
gfCNCPoint1[28444] = {X 153.5310, Y 45.9591, Z -2.1667, A 0.000, B 0.000, C 0.000 }
gfCNCPoint1[28445] = {X 153.2186, Y 46.8306, Z -2.1667, A 0.000, B 0.000, C 0.000 }
gfCNCPoint1[28446] = {X 152.7212, Y 47.6115, Z -2.1667, A 0.000, B 0.000, C 0.000 }
gfCNCPoint1[28447] = {X 152.0634, Y 48.2631, Z -2.1667, A 0.000, B 0.000, C 0.000 }
gfCNCPoint1[28448] = {X 151.2778, Y 48.7530, Z -2.1667, A 0.000, B 0.000, C 0.000 }
gfCNCPoint1[28449] = {X 150.4032, Y 49.0570, Z -2.1667, A 0.000, B 0.000, C 0.000 }
gfCNCPoint1[28450] = {X 149.4831, Y 49.1600, Z -2.1667, A 0.000, B 0.000, C 0.000 }
gfCNCPoint1[28451] = {X 143.0396, Y 49.1600, Z -2.1667, A 0.000, B 0.000, C 0.000 }
gfCNCPoint1[28452] = {X 142.1185, Y 49.0567, Z -2.1667, A 0.000, B 0.000, C 0.000 }
gfCNCPoint1[28453] = {X 141.2432, Y 48.7521, Z -2.1667, A 0.000, B 0.000, C 0.000 }
gfCNCPoint1[28454] = {X 140.4570, Y 48.2612, Z -2.1667, A 0.000, B 0.000, C 0.000 }
gfCNCPoint1[28455] = {X 139.7990, Y 47.6084, Z -2.1667, A 0.000, B 0.000, C 0.000 }
gfCNCPoint1[28456] = {X 139.3019, Y 46.8261, Z -2.1667, A 0.000, B 0.000, C 0.000 }
gfCNCPoint1[28457] = {X 138.9903, Y 45.9532, Z -2.1667, A 0.000, B 0.000, C 0.000 }
gfCNCPoint1[28458] = {X 138.8798, Y 45.0329, Z -2.1667, A 0.000, B 0.000, C 0.000 }
gfCNCPoint1[28459] = {X 138.8800, Y 44.1516, Z -2.1667, A 0.000, B 0.000, C 0.000 }
gfCNCPoint1[28460] = {X 138.9906, Y 43.2545, Z -2.1667, A 0.000, B 0.000, C 0.000 }
gfCNCPoint1[28461] = {X 139.2922, Y 42.4026, Z -2.1667, A 0.000, B 0.000, C 0.000 }
gfCNCPoint1[28462] = {X 139.7708, Y 41.6358, Z -2.1667, A 0.000, B 0.000, C 0.000 }
gfCNCPoint1[28463] = {X 140.4036, Y 40.9906, Z -2.1667, A 0.000, B 0.000, C 0.000 }
gfCNCPoint1[28464] = {X 140.4036, Y 30.3962, Z -2.1667, A 0.000, B 0.000, C 0.000 }
gfCNCPoint1[28465] = {X 136.4036, Y 30.3962, Z -2.1667, A 0.000, B 0.000, C 0.000 }
gfCNCPoint1[28466] = {X 140.4836, Y 30.3962, Z -2.1667, A 0.000, B 0.000, C 0.000 }
gfCNCPoint1[28467] = {X 140.4836, Y 19.6368, Z -2.1667, A 0.000, B 0.000, C 0.000 }
gfCNCPoint1[28468] = {X 137.2908, Y 19.6359, Z -2.1667, A 0.000, B 0.000, C 0.000 }
gfCNCPoint1[28469] = {X 137.2218, Y 19.7475, Z -2.1667, A 0.000, B 0.000, C 0.000 }
gfCNCPoint1[28470] = {X 136.5756, Y 20.4907, Z -2.1667, A 0.000, B 0.000, C 0.000 }
gfCNCPoint1[28471] = {X 135.7702, Y 21.0573, Z -2.1667, A 0.000, B 0.000, C 0.000 }
gfCNCPoint1[28472] = {X 134.8524, Y 21.4145, Z -2.1667, A 0.000, B 0.000, C 0.000 }
gfCNCPoint1[28473] = {X 133.8758, Y 21.5414, Z -2.1667, A 0.000, B 0.000, C 0.000 }
gfCNCPoint1[28474] = {X 133.2006, Y 21.5415, Z -2.1667, A 0.000, B 0.000, C 0.000 }
gfCNCPoint1[28475] = {X 132.2928, Y 21.4392, Z -2.1667, A 0.000, B 0.000, C 0.000 }
gfCNCPoint1[28476] = {X 131.4304, Y 21.1375, Z -2.1667, A 0.000, B 0.000, C 0.000 }
gfCNCPoint1[28477] = {X 130.6568, Y 20.6514, Z -2.1667, A 0.000, B 0.000, C 0.000 }
gfCNCPoint1[28478] = {X 130.0108, Y 20.0054, Z -2.1667, A 0.000, B 0.000, C 0.000 }
gfCNCPoint1[28479] = {X 129.5247, Y 19.2318, Z -2.1667, A 0.000, B 0.000, C 0.000 }
gfCNCPoint1[28480] = {X 129.2229, Y 18.3694, Z -2.1667, A 0.000, B 0.000, C 0.000 }
gfCNCPoint1[28481] = {X 129.1206, Y 17.4615, Z -2.1667, A 0.000, B 0.000, C 0.000 }
gfCNCPoint1[28482] = {X 129.1206, Y 10.4835, Z -2.1667, A 0.000, B 0.000, C 0.000 }
gfCNCPoint1[28483] = {X 129.2215, Y 9.5820, Z -2.1667, A 0.000, B 0.000, C 0.000 }
gfCNCPoint1[28484] = {X 129.5191, Y 8.7250, Z -2.1667, A 0.000, B 0.000, C 0.000 }
gfCNCPoint1[28485] = {X 129.9986, Y 7.9550, Z -2.1667, A 0.000, B 0.000, C 0.000 }
gfCNCPoint1[28486] = {X 130.6365, Y 7.3099, Z -2.1667, A 0.000, B 0.000, C 0.000 }
gfCNCPoint1[28487] = {X 131.4011, Y 6.8218, Z -2.1667, A 0.000, B 0.000, C 0.000 }
gfCNCPoint1[28488] = {X 132.2547, Y 6.5147, Z -2.1667, A 0.000, B 0.000, C 0.000 }
gfCNCPoint1[28489] = {X 133.1551, Y 6.4038, Z -2.1667, A 0.000, B 0.000, C 0.000 }
gfCNCPoint1[28490] = {X 133.8841, Y 6.4037, Z -2.1667, A 0.000, B 0.000, C 0.000 }
gfCNCPoint1[28491] = {X 134.6876, Y 6.4920, Z -2.1667, A 0.000, B 0.000, C 0.000 }
gfCNCPoint1[28492] = {X 135.4578, Y 6.7370, Z -2.1667, A 0.000, B 0.000, C 0.000 }
gfCNCPoint1[28493] = {X 136.1647, Y 7.1290, Z -2.1667, A 0.000, B 0.000, C 0.000 }
gfCNCPoint1[28494] = {X 136.7804, Y 7.6526, Z -2.1667, A 0.000, B 0.000, C 0.000 }
gfCNCPoint1[28495] = {X 137.2808, Y 8.2874, Z -2.1667, A 0.000, B 0.000, C 0.000 }
gfCNCPoint1[28496] = {X 155.2412, Y 8.2885, Z -2.1667, A 0.000, B 0.000, C 0.000 }
gfCNCPoint1[28497] = {X 155.2866, Y 8.2189, Z -2.1667, A 0.000, B 0.000, C 0.000 }
gfCNCPoint1[28498] = {X 155.3334, Y 8.1503, Z -2.1667, A 0.000, B 0.000, C 0.000 }
gfCNCPoint1[28499] = {X 155.9785, Y 7.4264, Z -2.1667, A 0.000, B 0.000, C 0.000 }
gfCNCPoint1[28500] = {X 156.7763, Y 6.8751, Z -2.1667, A 0.000, B 0.000, C 0.000 }
gfCNCPoint1[28501] = {X 157.6816, Y 6.5277, Z -2.1667, A 0.000, B 0.000, C 0.000 }
gfCNCPoint1[28502] = {X 158.6434, Y 6.4037, Z -2.1667, A 0.000, B 0.000, C 0.000 }
gfCNCPoint1[28503] = {X 159.3750, Y 6.4039, Z -2.1667, A 0.000, B 0.000, C 0.000 }
gfCNCPoint1[28504] = {X 160.2741, Y 6.5161, Z -2.1667, A 0.000, B 0.000, C 0.000 }
gfCNCPoint1[28505] = {X 161.1263, Y 6.8241, Z -2.1667, A 0.000, B 0.000, C 0.000 }
gfCNCPoint1[28506] = {X 161.8895, Y 7.3126, Z -2.1667, A 0.000, B 0.000, C 0.000 }
gfCNCPoint1[28507] = {X 162.5260, Y 7.9574, Z -2.1667, A 0.000, B 0.000, C 0.000 }
gfCNCPoint1[28508] = {X 163.0046, Y 8.7269, Z -2.1667, A 0.000, B 0.000, C 0.000 }
gfCNCPoint1[28509] = {X 163.3015, Y 9.5830, Z -2.1667, A 0.000, B 0.000, C 0.000 }
gfCNCPoint1[28510] = {X 163.4021, Y 10.4835, Z -2.1667, A 0.000, B 0.000, C 0.000 }
gfCNCPoint1[28511] = {X 163.4021, Y 17.4615, Z -2.1667, A 0.000, B 0.000, C 0.000 }
gfCNCPoint1[28512] = {X 163.3015, Y 18.3621, Z -2.1667, A 0.000, B 0.000, C 0.000 }
gfCNCPoint1[28513] = {X 163.0046, Y 19.2182, Z -2.1667, A 0.000, B 0.000, C 0.000 }
gfCNCPoint1[28514] = {X 162.5260, Y 19.9876, Z -2.1667, A 0.000, B 0.000, C 0.000 }
gfCNCPoint1[28515] = {X 161.8895, Y 20.6325, Z -2.1667, A 0.000, B 0.000, C 0.000 }
gfCNCPoint1[28516] = {X 161.1263, Y 21.1209, Z -2.1667, A 0.000, B 0.000, C 0.000 }
gfCNCPoint1[28517] = {X 160.2741, Y 21.4289, Z -2.1667, A 0.000, B 0.000, C 0.000 }
gfCNCPoint1[28518] = {X 159.3750, Y 21.5412, Z -2.1667, A 0.000, B 0.000, C 0.000 }
gfCNCPoint1[28519] = {X 158.6802, Y 21.5415, Z -2.1667, A 0.000, B 0.000, C 0.000 }
gfCNCPoint1[28520] = {X 157.8634, Y 21.4556, Z -2.1667, A 0.000, B 0.000, C 0.000 }
gfCNCPoint1[28521] = {X 157.0799, Y 21.2094, Z -2.1667, A 0.000, B 0.000, C 0.000 }
gfCNCPoint1[28522] = {X 156.3609, Y 20.8126, Z -2.1667, A 0.000, B 0.000, C 0.000 }
gfCNCPoint1[28523] = {X 155.7348, Y 20.2811, Z -2.1667, A 0.000, B 0.000, C 0.000 }
gfCNCPoint1[28524] = {X 155.2267, Y 19.6359, Z -2.1667, A 0.000, B 0.000, C 0.000 }
gfCNCPoint1[28525] = {X 152.0358, Y 19.6375, Z -2.1667, A 0.000, B 0.000, C 0.000 }
gfCNCPoint1[28526] = {X 152.0341, Y 40.9684, Z -2.1667, A 0.000, B 0.000, C 0.000 }
gfCNCPoint1[28527] = {X 152.5609, Y 41.5355, Z -2.1667, A 0.000, B 0.000, C 0.000 }
gfCNCPoint1[28528] = {X 152.6496, Y 41.6414, Z -2.1667, A 0.000, B 0.000, C 0.000 }
gfCNCPoint1[28529] = {X 153.1453, Y 42.4208, Z -2.1667, A 0.000, B 0.000, C 0.000 }
gfCNCPoint1[28530] = {X 153.4550, Y 43.2911, Z -2.1667, A 0.000, B 0.000, C 0.000 }
gfCNCPoint1[28531] = {X 153.5631, Y 44.2085, Z -2.1667, A 0.000, B 0.000, C 0.000 }
gfCNCPoint1[28532] = {X 153.5629, Y 45.0392, Z -2.1667, A 0.000, B 0.000, C 0.000 }
gfCNCPoint1[28533] = {X 153.4532, Y 45.9406, Z -2.1667, A 0.000, B 0.000, C 0.000 }
gfCNCPoint1[28534] = {X 153.1468, Y 46.7954, Z -2.1667, A 0.000, B 0.000, C 0.000 }
gfCNCPoint1[28535] = {X 152.6589, Y 47.5613, Z -2.1667, A 0.000, B 0.000, C 0.000 }
gfCNCPoint1[28536] = {X 152.0138, Y 48.2003, Z -2.1667, A 0.000, B 0.000, C 0.000 }
gfCNCPoint1[28537] = {X 151.2432, Y 48.6808, Z -2.1667, A 0.000, B 0.000, C 0.000 }
gfCNCPoint1[28538] = {X 150.3855, Y 48.9789, Z -2.1667, A 0.000, B 0.000, C 0.000 }
gfCNCPoint1[28539] = {X 149.4831, Y 49.0800, Z -2.1667, A 0.000, B 0.000, C 0.000 }
gfCNCPoint1[28540] = {X 143.0396, Y 49.0800, Z -2.1667, A 0.000, B 0.000, C 0.000 }
gfCNCPoint1[28541] = {X 142.1362, Y 48.9787, Z -2.1667, A 0.000, B 0.000, C 0.000 }
gfCNCPoint1[28542] = {X 141.2777, Y 48.6799, Z -2.1667, A 0.000, B 0.000, C 0.000 }
gfCNCPoint1[28543] = {X 140.5066, Y 48.1985, Z -2.1667, A 0.000, B 0.000, C 0.000 }
gfCNCPoint1[28544] = {X 139.8613, Y 47.5582, Z -2.1667, A 0.000, B 0.000, C 0.000 }
gfCNCPoint1[28545] = {X 139.3737, Y 46.7910, Z -2.1667, A 0.000, B 0.000, C 0.000 }
gfCNCPoint1[28546] = {X 139.0682, Y 45.9349, Z -2.1667, A 0.000, B 0.000, C 0.000 }
gfCNCPoint1[28547] = {X 138.9598, Y 45.0323, Z -2.1667, A 0.000, B 0.000, C 0.000 }
gfCNCPoint1[28548] = {X 138.9600, Y 44.1527, Z -2.1667, A 0.000, B 0.000, C 0.000 }
gfCNCPoint1[28549] = {X 139.0706, Y 43.2637, Z -2.1667, A 0.000, B 0.000, C 0.000 }
gfCNCPoint1[28550] = {X 139.3725, Y 42.4203, Z -2.1667, A 0.000, B 0.000, C 0.000 }
gfCNCPoint1[28551] = {X 139.8512, Y 41.6631, Z -2.1667, A 0.000, B 0.000, C 0.000 }
gfCNCPoint1[28552] = {X 140.4836, Y 41.0287, Z -2.1667, A 0.000, B 0.000, C 0.000 }
gfCNCPoint1[28553] = {X 140.4836, Y 30.3962, Z -2.1667, A 0.000, B 0.000, C 0.000 }
gfCNCPoint1[28554] = {X 136.4836, Y 30.3962, Z -2.1667, A 0.000, B 0.000, C 0.000 }
gfCNCPoint1[28555] = {X 140.5636, Y 30.3962, Z -2.1667, A 0.000, B 0.000, C 0.000 }
gfCNCPoint1[28556] = {X 140.5636, Y 19.9567, Z -2.1667, A 0.000, B 0.000, C 0.000 }
gfCNCPoint1[28557] = {X 140.5650, Y 19.5568, Z -2.1667, A 0.000, B 0.000, C 0.000 }
gfCNCPoint1[28558] = {X 137.2663, Y 19.5559, Z -2.1667, A 0.000, B 0.000, C 0.000 }
gfCNCPoint1[28559] = {X 137.2436, Y 19.5600, Z -2.1667, A 0.000, B 0.000, C 0.000 }
gfCNCPoint1[28560] = {X 137.1374, Y 19.7292, Z -2.1667, A 0.000, B 0.000, C 0.000 }
gfCNCPoint1[28561] = {X 136.4979, Y 20.4528, Z -2.1667, A 0.000, B 0.000, C 0.000 }
gfCNCPoint1[28562] = {X 135.7036, Y 21.0021, Z -2.1667, A 0.000, B 0.000, C 0.000 }
gfCNCPoint1[28563] = {X 134.8008, Y 21.3450, Z -2.1667, A 0.000, B 0.000, C 0.000 }
gfCNCPoint1[28564] = {X 133.8421, Y 21.4615, Z -2.1667, A 0.000, B 0.000, C 0.000 }
gfCNCPoint1[28565] = {X 133.2006, Y 21.4615, Z -2.1667, A 0.000, B 0.000, C 0.000 }
gfCNCPoint1[28566] = {X 132.3106, Y 21.3612, Z -2.1667, A 0.000, B 0.000, C 0.000 }
gfCNCPoint1[28567] = {X 131.4651, Y 21.0654, Z -2.1667, A 0.000, B 0.000, C 0.000 }
gfCNCPoint1[28568] = {X 130.7067, Y 20.5889, Z -2.1667, A 0.000, B 0.000, C 0.000 }
gfCNCPoint1[28569] = {X 130.0733, Y 19.9555, Z -2.1667, A 0.000, B 0.000, C 0.000 }
gfCNCPoint1[28570] = {X 129.5968, Y 19.1971, Z -2.1667, A 0.000, B 0.000, C 0.000 }
gfCNCPoint1[28571] = {X 129.3009, Y 18.3516, Z -2.1667, A 0.000, B 0.000, C 0.000 }
gfCNCPoint1[28572] = {X 129.2006, Y 17.4615, Z -2.1667, A 0.000, B 0.000, C 0.000 }
gfCNCPoint1[28573] = {X 129.2006, Y 10.4835, Z -2.1667, A 0.000, B 0.000, C 0.000 }
gfCNCPoint1[28574] = {X 129.3009, Y 9.5934, Z -2.1667, A 0.000, B 0.000, C 0.000 }
gfCNCPoint1[28575] = {X 129.5968, Y 8.7480, Z -2.1667, A 0.000, B 0.000, C 0.000 }
gfCNCPoint1[28576] = {X 130.0733, Y 7.9895, Z -2.1667, A 0.000, B 0.000, C 0.000 }
gfCNCPoint1[28577] = {X 130.7067, Y 7.3562, Z -2.1667, A 0.000, B 0.000, C 0.000 }
gfCNCPoint1[28578] = {X 131.4651, Y 6.8796, Z -2.1667, A 0.000, B 0.000, C 0.000 }
gfCNCPoint1[28579] = {X 132.3106, Y 6.5838, Z -2.1667, A 0.000, B 0.000, C 0.000 }
gfCNCPoint1[28580] = {X 133.2007, Y 6.4835, Z -2.1667, A 0.000, B 0.000, C 0.000 }
gfCNCPoint1[28581] = {X 133.8833, Y 6.4837, Z -2.1667, A 0.000, B 0.000, C 0.000 }
gfCNCPoint1[28582] = {X 134.6795, Y 6.5721, Z -2.1667, A 0.000, B 0.000, C 0.000 }
gfCNCPoint1[28583] = {X 135.4422, Y 6.8174, Z -2.1667, A 0.000, B 0.000, C 0.000 }
gfCNCPoint1[28584] = {X 136.1407, Y 7.2097, Z -2.1667, A 0.000, B 0.000, C 0.000 }
gfCNCPoint1[28585] = {X 136.7469, Y 7.7334, Z -2.1667, A 0.000, B 0.000, C 0.000 }
gfCNCPoint1[28586] = {X 137.2367, Y 8.3674, Z -2.1667, A 0.000, B 0.000, C 0.000 }
gfCNCPoint1[28587] = {X 155.2276, Y 8.3674, Z -2.1667, A 0.000, B 0.000, C 0.000 }
gfCNCPoint1[28588] = {X 155.2814, Y 8.3748, Z -2.1667, A 0.000, B 0.000, C 0.000 }
gfCNCPoint1[28589] = {X 155.3390, Y 8.2846, Z -2.1667, A 0.000, B 0.000, C 0.000 }
gfCNCPoint1[28590] = {X 155.3990, Y 8.1961, Z -2.1667, A 0.000, B 0.000, C 0.000 }
gfCNCPoint1[28591] = {X 156.0383, Y 7.4803, Z -2.1667, A 0.000, B 0.000, C 0.000 }
gfCNCPoint1[28592] = {X 156.8298, Y 6.9374, Z -2.1667, A 0.000, B 0.000, C 0.000 }
gfCNCPoint1[28593] = {X 157.7278, Y 6.5986, Z -2.1667, A 0.000, B 0.000, C 0.000 }
gfCNCPoint1[28594] = {X 158.6806, Y 6.4835, Z -2.1667, A 0.000, B 0.000, C 0.000 }
gfCNCPoint1[28595] = {X 159.3739, Y 6.4839, Z -2.1667, A 0.000, B 0.000, C 0.000 }
gfCNCPoint1[28596] = {X 160.2554, Y 6.5939, Z -2.1667, A 0.000, B 0.000, C 0.000 }
gfCNCPoint1[28597] = {X 161.0909, Y 6.8959, Z -2.1667, A 0.000, B 0.000, C 0.000 }
gfCNCPoint1[28598] = {X 161.8391, Y 7.3747, Z -2.1667, A 0.000, B 0.000, C 0.000 }
gfCNCPoint1[28599] = {X 162.4632, Y 8.0070, Z -2.1667, A 0.000, B 0.000, C 0.000 }
gfCNCPoint1[28600] = {X 162.9324, Y 8.7613, Z -2.1667, A 0.000, B 0.000, C 0.000 }
gfCNCPoint1[28601] = {X 163.2234, Y 9.6007, Z -2.1667, A 0.000, B 0.000, C 0.000 }
gfCNCPoint1[28602] = {X 163.3221, Y 10.4835, Z -2.1667, A 0.000, B 0.000, C 0.000 }
gfCNCPoint1[28603] = {X 163.3221, Y 17.4615, Z -2.1667, A 0.000, B 0.000, C 0.000 }
gfCNCPoint1[28604] = {X 163.2218, Y 18.3516, Z -2.1667, A 0.000, B 0.000, C 0.000 }
gfCNCPoint1[28605] = {X 162.9260, Y 19.1971, Z -2.1667, A 0.000, B 0.000, C 0.000 }
gfCNCPoint1[28606] = {X 162.4494, Y 19.9555, Z -2.1667, A 0.000, B 0.000, C 0.000 }
gfCNCPoint1[28607] = {X 161.8160, Y 20.5889, Z -2.1667, A 0.000, B 0.000, C 0.000 }
gfCNCPoint1[28608] = {X 161.0576, Y 21.0654, Z -2.1667, A 0.000, B 0.000, C 0.000 }
gfCNCPoint1[28609] = {X 160.2121, Y 21.3613, Z -2.1667, A 0.000, B 0.000, C 0.000 }
gfCNCPoint1[28610] = {X 159.3221, Y 21.4615, Z -2.1667, A 0.000, B 0.000, C 0.000 }
gfCNCPoint1[28611] = {X 158.6806, Y 21.4615, Z -2.1667, A 0.000, B 0.000, C 0.000 }
gfCNCPoint1[28612] = {X 157.8711, Y 21.3755, Z -2.1667, A 0.000, B 0.000, C 0.000 }
gfCNCPoint1[28613] = {X 157.0953, Y 21.1289, Z -2.1667, A 0.000, B 0.000, C 0.000 }
gfCNCPoint1[28614] = {X 156.3848, Y 20.7318, Z -2.1667, A 0.000, B 0.000, C 0.000 }
gfCNCPoint1[28615] = {X 155.7682, Y 20.2003, Z -2.1667, A 0.000, B 0.000, C 0.000 }
gfCNCPoint1[28616] = {X 155.2709, Y 19.5559, Z -2.1667, A 0.000, B 0.000, C 0.000 }
gfCNCPoint1[28617] = {X 151.9558, Y 19.5575, Z -2.1667, A 0.000, B 0.000, C 0.000 }
gfCNCPoint1[28618] = {X 151.9541, Y 40.9999, Z -2.1667, A 0.000, B 0.000, C 0.000 }
gfCNCPoint1[28619] = {X 152.5009, Y 41.5885, Z -2.1667, A 0.000, B 0.000, C 0.000 }
gfCNCPoint1[28620] = {X 152.5878, Y 41.6922, Z -2.1667, A 0.000, B 0.000, C 0.000 }
gfCNCPoint1[28621] = {X 153.0736, Y 42.4564, Z -2.1667, A 0.000, B 0.000, C 0.000 }
gfCNCPoint1[28622] = {X 153.3772, Y 43.3096, Z -2.1667, A 0.000, B 0.000, C 0.000 }
gfCNCPoint1[28623] = {X 153.4831, Y 44.2089, Z -2.1667, A 0.000, B 0.000, C 0.000 }
gfCNCPoint1[28624] = {X 153.4829, Y 45.0384, Z -2.1667, A 0.000, B 0.000, C 0.000 }
gfCNCPoint1[28625] = {X 153.3753, Y 45.9222, Z -2.1667, A 0.000, B 0.000, C 0.000 }
gfCNCPoint1[28626] = {X 153.0750, Y 46.7602, Z -2.1667, A 0.000, B 0.000, C 0.000 }
gfCNCPoint1[28627] = {X 152.5967, Y 47.5111, Z -2.1667, A 0.000, B 0.000, C 0.000 }
gfCNCPoint1[28628] = {X 151.9642, Y 48.1376, Z -2.1667, A 0.000, B 0.000, C 0.000 }
gfCNCPoint1[28629] = {X 151.2087, Y 48.6086, Z -2.1667, A 0.000, B 0.000, C 0.000 }
gfCNCPoint1[28630] = {X 150.3678, Y 48.9009, Z -2.1667, A 0.000, B 0.000, C 0.000 }
gfCNCPoint1[28631] = {X 149.4831, Y 49.0000, Z -2.1667, A 0.000, B 0.000, C 0.000 }
gfCNCPoint1[28632] = {X 143.0396, Y 49.0000, Z -2.1667, A 0.000, B 0.000, C 0.000 }
gfCNCPoint1[28633] = {X 142.1495, Y 48.8997, Z -2.1667, A 0.000, B 0.000, C 0.000 }
gfCNCPoint1[28634] = {X 141.3041, Y 48.6039, Z -2.1667, A 0.000, B 0.000, C 0.000 }
gfCNCPoint1[28635] = {X 140.5457, Y 48.1273, Z -2.1667, A 0.000, B 0.000, C 0.000 }
gfCNCPoint1[28636] = {X 139.9123, Y 47.4939, Z -2.1667, A 0.000, B 0.000, C 0.000 }
gfCNCPoint1[28637] = {X 139.4357, Y 46.7355, Z -2.1667, A 0.000, B 0.000, C 0.000 }
gfCNCPoint1[28638] = {X 139.1399, Y 45.8900, Z -2.1667, A 0.000, B 0.000, C 0.000 }
gfCNCPoint1[28639] = {X 139.0396, Y 45.0000, Z -2.1667, A 0.000, B 0.000, C 0.000 }
gfCNCPoint1[28640] = {X 139.0400, Y 44.1538, Z -2.1667, A 0.000, B 0.000, C 0.000 }
gfCNCPoint1[28641] = {X 139.1506, Y 43.2730, Z -2.1667, A 0.000, B 0.000, C 0.000 }
gfCNCPoint1[28642] = {X 139.4528, Y 42.4382, Z -2.1667, A 0.000, B 0.000, C 0.000 }
gfCNCPoint1[28643] = {X 139.9317, Y 41.6907, Z -2.1667, A 0.000, B 0.000, C 0.000 }
gfCNCPoint1[28644] = {X 140.5636, Y 41.0672, Z -2.1667, A 0.000, B 0.000, C 0.000 }
gfCNCPoint1[28645] = {X 140.5636, Y 30.3962, Z -2.1667, A 0.000, B 0.000, C 0.000 }
gfCNCPoint1[28646] = {X 136.4836, Y 30.3962, Z -2.1667, A 0.000, B 0.000, C 0.000 }
gfCNCPoint1[28647] = {X 136.4836, Y 30.3962, Z 0.8333, A 0.000, B 0.000, C 0.000 }
gfCNCPoint1[28648] = {X 136.4836, Y 30.3962, Z 11.0000, A 0.000, B 0.000, C 0.000 }
gfCNCPoint1[28649] = {X 137.6638, Y 74.8935, Z 11.0000, A 0.000, B 0.000, C 0.000 }
gfCNCPoint1[28650] = {X 137.6638, Y 74.8935, Z 0.8333, A 0.000, B 0.000, C 0.000 }
gfCNCPoint1[28651] = {X 137.6638, Y 74.8935, Z -2.1667, A 0.000, B 0.000, C 0.000 }
gfCNCPoint1[28652] = {X 140.6805, Y 77.6405, Z -2.1667, A 0.000, B 0.000, C 0.000 }
gfCNCPoint1[28653] = {X 155.6328, Y 61.2208, Z -2.1667, A 0.000, B 0.000, C 0.000 }
gfCNCPoint1[28654] = {X 155.2776, Y 60.5149, Z -2.1667, A 0.000, B 0.000, C 0.000 }
gfCNCPoint1[28655] = {X 155.0569, Y 59.7561, Z -2.1667, A 0.000, B 0.000, C 0.000 }
gfCNCPoint1[28656] = {X 154.9781, Y 58.9697, Z -2.1667, A 0.000, B 0.000, C 0.000 }
gfCNCPoint1[28657] = {X 154.9780, Y 58.0000, Z -2.1667, A 0.000, B 0.000, C 0.000 }
gfCNCPoint1[28658] = {X 155.0863, Y 57.0387, Z -2.1667, A 0.000, B 0.000, C 0.000 }
gfCNCPoint1[28659] = {X 155.4058, Y 56.1256, Z -2.1667, A 0.000, B 0.000, C 0.000 }
gfCNCPoint1[28660] = {X 155.9204, Y 55.3065, Z -2.1667, A 0.000, B 0.000, C 0.000 }
gfCNCPoint1[28661] = {X 156.6045, Y 54.6225, Z -2.1667, A 0.000, B 0.000, C 0.000 }
gfCNCPoint1[28662] = {X 157.4236, Y 54.1078, Z -2.1667, A 0.000, B 0.000, C 0.000 }
gfCNCPoint1[28663] = {X 158.3367, Y 53.7883, Z -2.1667, A 0.000, B 0.000, C 0.000 }
gfCNCPoint1[28664] = {X 159.2980, Y 53.6800, Z -2.1667, A 0.000, B 0.000, C 0.000 }
gfCNCPoint1[28665] = {X 178.5335, Y 53.6800, Z -2.1667, A 0.000, B 0.000, C 0.000 }
gfCNCPoint1[28666] = {X 179.4948, Y 53.7883, Z -2.1667, A 0.000, B 0.000, C 0.000 }
gfCNCPoint1[28667] = {X 180.4079, Y 54.1078, Z -2.1667, A 0.000, B 0.000, C 0.000 }
gfCNCPoint1[28668] = {X 181.2270, Y 54.6225, Z -2.1667, A 0.000, B 0.000, C 0.000 }
gfCNCPoint1[28669] = {X 181.9110, Y 55.3065, Z -2.1667, A 0.000, B 0.000, C 0.000 }
gfCNCPoint1[28670] = {X 182.4257, Y 56.1256, Z -2.1667, A 0.000, B 0.000, C 0.000 }
gfCNCPoint1[28671] = {X 182.7452, Y 57.0387, Z -2.1667, A 0.000, B 0.000, C 0.000 }
gfCNCPoint1[28672] = {X 182.8535, Y 58.0000, Z -2.1667, A 0.000, B 0.000, C 0.000 }
gfCNCPoint1[28673] = {X 182.8535, Y 58.9342, Z -2.1667, A 0.000, B 0.000, C 0.000 }
gfCNCPoint1[28674] = {X 182.7808, Y 59.7235, Z -2.1667, A 0.000, B 0.000, C 0.000 }
gfCNCPoint1[28675] = {X 182.5650, Y 60.4863, Z -2.1667, A 0.000, B 0.000, C 0.000 }
gfCNCPoint1[28676] = {X 182.2135, Y 61.1968, Z -2.1667, A 0.000, B 0.000, C 0.000 }
gfCNCPoint1[28677] = {X 209.4775, Y 90.9539, Z -2.1667, A 0.000, B 0.000, C 0.000 }
gfCNCPoint1[28678] = {X 210.1357, Y 91.6216, Z -2.1667, A 0.000, B 0.000, C 0.000 }
gfCNCPoint1[28679] = {X 210.8407, Y 92.2396, Z -2.1667, A 0.000, B 0.000, C 0.000 }
gfCNCPoint1[28680] = {X 211.1142, Y 92.4127, Z -2.1667, A 0.000, B 0.000, C 0.000 }
gfCNCPoint1[28681] = {X 211.4210, Y 92.5162, Z -2.1667, A 0.000, B 0.000, C 0.000 }
gfCNCPoint1[28682] = {X 213.4038, Y 92.8255, Z -2.1667, A 0.000, B 0.000, C 0.000 }
gfCNCPoint1[28683] = {X 214.4545, Y 92.7368, Z -2.1667, A 0.000, B 0.000, C 0.000 }
gfCNCPoint1[28684] = {X 215.5072, Y 92.6766, Z -2.1667, A 0.000, B 0.000, C 0.000 }
gfCNCPoint1[28685] = {X 216.1772, Y 92.6031, Z -2.1667, A 0.000, B 0.000, C 0.000 }
gfCNCPoint1[28686] = {X 216.8225, Y 92.4081, Z -2.1667, A 0.000, B 0.000, C 0.000 }
gfCNCPoint1[28687] = {X 217.4211, Y 92.0980, Z -2.1667, A 0.000, B 0.000, C 0.000 }
gfCNCPoint1[28688] = {X 222.9613, Y 88.5226, Z -2.1667, A 0.000, B 0.000, C 0.000 }
gfCNCPoint1[28689] = {X 245.8291, Y 73.8995, Z -2.1667, A 0.000, B 0.000, C 0.000 }
gfCNCPoint1[28690] = {X 221.6305, Y 64.4027, Z -2.1667, A 0.000, B 0.000, C 0.000 }
gfCNCPoint1[28691] = {X 219.8632, Y 63.8112, Z -2.1667, A 0.000, B 0.000, C 0.000 }
gfCNCPoint1[28692] = {X 218.0398, Y 63.4258, Z -2.1667, A 0.000, B 0.000, C 0.000 }
gfCNCPoint1[28693] = {X 216.1843, Y 63.2516, Z -2.1667, A 0.000, B 0.000, C 0.000 }
gfCNCPoint1[28694] = {X 215.2524, Y 63.1173, Z -2.1667, A 0.000, B 0.000, C 0.000 }
gfCNCPoint1[28695] = {X 214.3717, Y 62.7843, Z -2.1667, A 0.000, B 0.000, C 0.000 }
gfCNCPoint1[28696] = {X 213.5841, Y 62.2685, Z -2.1667, A 0.000, B 0.000, C 0.000 }
gfCNCPoint1[28697] = {X 212.9270, Y 61.5942, Z -2.1667, A 0.000, B 0.000, C 0.000 }
gfCNCPoint1[28698] = {X 212.4315, Y 60.7937, Z -2.1667, A 0.000, B 0.000, C 0.000 }
gfCNCPoint1[28699] = {X 212.1213, Y 59.9048, Z -2.1667, A 0.000, B 0.000, C 0.000 }
gfCNCPoint1[28700] = {X 212.0110, Y 58.9697, Z -2.1667, A 0.000, B 0.000, C 0.000 }
gfCNCPoint1[28701] = {X 212.0108, Y 58.0000, Z -2.1667, A 0.000, B 0.000, C 0.000 }
gfCNCPoint1[28702] = {X 212.1191, Y 57.0387, Z -2.1667, A 0.000, B 0.000, C 0.000 }
gfCNCPoint1[28703] = {X 212.4386, Y 56.1256, Z -2.1667, A 0.000, B 0.000, C 0.000 }
gfCNCPoint1[28704] = {X 212.9533, Y 55.3065, Z -2.1667, A 0.000, B 0.000, C 0.000 }
gfCNCPoint1[28705] = {X 213.6373, Y 54.6225, Z -2.1667, A 0.000, B 0.000, C 0.000 }
gfCNCPoint1[28706] = {X 214.4564, Y 54.1078, Z -2.1667, A 0.000, B 0.000, C 0.000 }
gfCNCPoint1[28707] = {X 215.3695, Y 53.7883, Z -2.1667, A 0.000, B 0.000, C 0.000 }
gfCNCPoint1[28708] = {X 216.3308, Y 53.6800, Z -2.1667, A 0.000, B 0.000, C 0.000 }
gfCNCPoint1[28709] = {X 237.2617, Y 53.6800, Z -2.1667, A 0.000, B 0.000, C 0.000 }
gfCNCPoint1[28710] = {X 238.2230, Y 53.7883, Z -2.1667, A 0.000, B 0.000, C 0.000 }
gfCNCPoint1[28711] = {X 239.1361, Y 54.1078, Z -2.1667, A 0.000, B 0.000, C 0.000 }
gfCNCPoint1[28712] = {X 239.9552, Y 54.6225, Z -2.1667, A 0.000, B 0.000, C 0.000 }
gfCNCPoint1[28713] = {X 240.6392, Y 55.3065, Z -2.1667, A 0.000, B 0.000, C 0.000 }
gfCNCPoint1[28714] = {X 241.1539, Y 56.1256, Z -2.1667, A 0.000, B 0.000, C 0.000 }
gfCNCPoint1[28715] = {X 241.4734, Y 57.0387, Z -2.1667, A 0.000, B 0.000, C 0.000 }
gfCNCPoint1[28716] = {X 241.5817, Y 58.0000, Z -2.1667, A 0.000, B 0.000, C 0.000 }
gfCNCPoint1[28717] = {X 241.5817, Y 58.2329, Z -2.1667, A 0.000, B 0.000, C 0.000 }
gfCNCPoint1[28718] = {X 247.4883, Y 60.5356, Z -2.1667, A 0.000, B 0.000, C 0.000 }
gfCNCPoint1[28719] = {X 275.6338, Y 71.7030, Z -2.1667, A 0.000, B 0.000, C 0.000 }
gfCNCPoint1[28720] = {X 275.6344, Y 63.2124, Z -2.1667, A 0.000, B 0.000, C 0.000 }
gfCNCPoint1[28721] = {X 274.7827, Y 63.0034, Z -2.1667, A 0.000, B 0.000, C 0.000 }
gfCNCPoint1[28722] = {X 273.9906, Y 62.6267, Z -2.1667, A 0.000, B 0.000, C 0.000 }
gfCNCPoint1[28723] = {X 273.2910, Y 62.0978, Z -2.1667, A 0.000, B 0.000, C 0.000 }
gfCNCPoint1[28724] = {X 272.7127, Y 61.4384, Z -2.1667, A 0.000, B 0.000, C 0.000 }
gfCNCPoint1[28725] = {X 272.2794, Y 60.6759, Z -2.1667, A 0.000, B 0.000, C 0.000 }
gfCNCPoint1[28726] = {X 272.0091, Y 59.8415, Z -2.1667, A 0.000, B 0.000, C 0.000 }
gfCNCPoint1[28727] = {X 271.9128, Y 58.9697, Z -2.1667, A 0.000, B 0.000, C 0.000 }
gfCNCPoint1[28728] = {X 271.9127, Y 58.0000, Z -2.1667, A 0.000, B 0.000, C 0.000 }
gfCNCPoint1[28729] = {X 272.0210, Y 57.0387, Z -2.1667, A 0.000, B 0.000, C 0.000 }
gfCNCPoint1[28730] = {X 272.3405, Y 56.1256, Z -2.1667, A 0.000, B 0.000, C 0.000 }
gfCNCPoint1[28731] = {X 272.8552, Y 55.3065, Z -2.1667, A 0.000, B 0.000, C 0.000 }
gfCNCPoint1[28732] = {X 273.5392, Y 54.6225, Z -2.1667, A 0.000, B 0.000, C 0.000 }
gfCNCPoint1[28733] = {X 274.3583, Y 54.1078, Z -2.1667, A 0.000, B 0.000, C 0.000 }
gfCNCPoint1[28734] = {X 275.2714, Y 53.7883, Z -2.1667, A 0.000, B 0.000, C 0.000 }
gfCNCPoint1[28735] = {X 276.2327, Y 53.6800, Z -2.1667, A 0.000, B 0.000, C 0.000 }
gfCNCPoint1[28736] = {X 292.7731, Y 53.6800, Z -2.1667, A 0.000, B 0.000, C 0.000 }
gfCNCPoint1[28737] = {X 293.7344, Y 53.7883, Z -2.1667, A 0.000, B 0.000, C 0.000 }
gfCNCPoint1[28738] = {X 294.6475, Y 54.1078, Z -2.1667, A 0.000, B 0.000, C 0.000 }
gfCNCPoint1[28739] = {X 295.4666, Y 54.6225, Z -2.1667, A 0.000, B 0.000, C 0.000 }
gfCNCPoint1[28740] = {X 296.1506, Y 55.3065, Z -2.1667, A 0.000, B 0.000, C 0.000 }
gfCNCPoint1[28741] = {X 296.6653, Y 56.1256, Z -2.1667, A 0.000, B 0.000, C 0.000 }
gfCNCPoint1[28742] = {X 296.9848, Y 57.0387, Z -2.1667, A 0.000, B 0.000, C 0.000 }
gfCNCPoint1[28743] = {X 297.0931, Y 58.0000, Z -2.1667, A 0.000, B 0.000, C 0.000 }
gfCNCPoint1[28744] = {X 297.0931, Y 58.9352, Z -2.1667, A 0.000, B 0.000, C 0.000 }
gfCNCPoint1[28745] = {X 296.9708, Y 59.9431, Z -2.1667, A 0.000, B 0.000, C 0.000 }
gfCNCPoint1[28746] = {X 296.6174, Y 60.8949, Z -2.1667, A 0.000, B 0.000, C 0.000 }
gfCNCPoint1[28747] = {X 296.0525, Y 61.7385, Z -2.1667, A 0.000, B 0.000, C 0.000 }
gfCNCPoint1[28748] = {X 295.3070, Y 62.4277, Z -2.1667, A 0.000, B 0.000, C 0.000 }
gfCNCPoint1[28749] = {X 294.4216, Y 62.9246, Z -2.1667, A 0.000, B 0.000, C 0.000 }
gfCNCPoint1[28750] = {X 293.4449, Y 63.2021, Z -2.1667, A 0.000, B 0.000, C 0.000 }
gfCNCPoint1[28751] = {X 293.3718, Y 63.2250, Z -2.1667, A 0.000, B 0.000, C 0.000 }
gfCNCPoint1[28752] = {X 293.3841, Y 92.7821, Z -2.1667, A 0.000, B 0.000, C 0.000 }
gfCNCPoint1[28753] = {X 294.2366, Y 92.9995, Z -2.1667, A 0.000, B 0.000, C 0.000 }
gfCNCPoint1[28754] = {X 295.0279, Y 93.3838, Z -2.1667, A 0.000, B 0.000, C 0.000 }
gfCNCPoint1[28755] = {X 295.7258, Y 93.9194, Z -2.1667, A 0.000, B 0.000, C 0.000 }
gfCNCPoint1[28756] = {X 296.3017, Y 94.5844, Z -2.1667, A 0.000, B 0.000, C 0.000 }
gfCNCPoint1[28757] = {X 296.7322, Y 95.3516, Z -2.1667, A 0.000, B 0.000, C 0.000 }
gfCNCPoint1[28758] = {X 296.9996, Y 96.1897, Z -2.1667, A 0.000, B 0.000, C 0.000 }
gfCNCPoint1[28759] = {X 297.0931, Y 97.0644, Z -2.1667, A 0.000, B 0.000, C 0.000 }
gfCNCPoint1[28760] = {X 297.0931, Y 98.0000, Z -2.1667, A 0.000, B 0.000, C 0.000 }
gfCNCPoint1[28761] = {X 296.9848, Y 98.9613, Z -2.1667, A 0.000, B 0.000, C 0.000 }
gfCNCPoint1[28762] = {X 296.6653, Y 99.8744, Z -2.1667, A 0.000, B 0.000, C 0.000 }
gfCNCPoint1[28763] = {X 296.1506, Y 100.6935, Z -2.1667, A 0.000, B 0.000, C 0.000 }
gfCNCPoint1[28764] = {X 295.4666, Y 101.3775, Z -2.1667, A 0.000, B 0.000, C 0.000 }
gfCNCPoint1[28765] = {X 294.6475, Y 101.8922, Z -2.1667, A 0.000, B 0.000, C 0.000 }
gfCNCPoint1[28766] = {X 293.7344, Y 102.2117, Z -2.1667, A 0.000, B 0.000, C 0.000 }
gfCNCPoint1[28767] = {X 292.7731, Y 102.3200, Z -2.1667, A 0.000, B 0.000, C 0.000 }
gfCNCPoint1[28768] = {X 276.2327, Y 102.3200, Z -2.1667, A 0.000, B 0.000, C 0.000 }
gfCNCPoint1[28769] = {X 275.2714, Y 102.2117, Z -2.1667, A 0.000, B 0.000, C 0.000 }
gfCNCPoint1[28770] = {X 274.3583, Y 101.8922, Z -2.1667, A 0.000, B 0.000, C 0.000 }
gfCNCPoint1[28771] = {X 273.5392, Y 101.3775, Z -2.1667, A 0.000, B 0.000, C 0.000 }
gfCNCPoint1[28772] = {X 272.8552, Y 100.6935, Z -2.1667, A 0.000, B 0.000, C 0.000 }
gfCNCPoint1[28773] = {X 272.3405, Y 99.8744, Z -2.1667, A 0.000, B 0.000, C 0.000 }
gfCNCPoint1[28774] = {X 272.0210, Y 98.9613, Z -2.1667, A 0.000, B 0.000, C 0.000 }
gfCNCPoint1[28775] = {X 271.9127, Y 98.0000, Z -2.1667, A 0.000, B 0.000, C 0.000 }
gfCNCPoint1[28776] = {X 271.9127, Y 97.0659, Z -2.1667, A 0.000, B 0.000, C 0.000 }
gfCNCPoint1[28777] = {X 272.0026, Y 96.1891, Z -2.1667, A 0.000, B 0.000, C 0.000 }
gfCNCPoint1[28778] = {X 272.2686, Y 95.3488, Z -2.1667, A 0.000, B 0.000, C 0.000 }
gfCNCPoint1[28779] = {X 272.6996, Y 94.5800, Z -2.1667, A 0.000, B 0.000, C 0.000 }
gfCNCPoint1[28780] = {X 273.2777, Y 93.9147, Z -2.1667, A 0.000, B 0.000, C 0.000 }
gfCNCPoint1[28781] = {X 273.9788, Y 93.3805, Z -2.1667, A 0.000, B 0.000, C 0.000 }
gfCNCPoint1[28782] = {X 274.7737, Y 92.9998, Z -2.1667, A 0.000, B 0.000, C 0.000 }
gfCNCPoint1[28783] = {X 275.6294, Y 92.7883, Z -2.1667, A 0.000, B 0.000, C 0.000 }
gfCNCPoint1[28784] = {X 275.6294, Y 85.5950, Z -2.1667, A 0.000, B 0.000, C 0.000 }
gfCNCPoint1[28785] = {X 262.6395, Y 80.5029, Z -2.1667, A 0.000, B 0.000, C 0.000 }
gfCNCPoint1[28786] = {X 262.2760, Y 80.7317, Z -2.1667, A 0.000, B 0.000, C 0.000 }
gfCNCPoint1[28787] = {X 237.7959, Y 96.5879, Z -2.1667, A 0.000, B 0.000, C 0.000 }
gfCNCPoint1[28788] = {X 237.7998, Y 97.0646, Z -2.1667, A 0.000, B 0.000, C 0.000 }
gfCNCPoint1[28789] = {X 237.7998, Y 98.0000, Z -2.1667, A 0.000, B 0.000, C 0.000 }
gfCNCPoint1[28790] = {X 237.6915, Y 98.9613, Z -2.1667, A 0.000, B 0.000, C 0.000 }
gfCNCPoint1[28791] = {X 237.3720, Y 99.8744, Z -2.1667, A 0.000, B 0.000, C 0.000 }
gfCNCPoint1[28792] = {X 236.8573, Y 100.6935, Z -2.1667, A 0.000, B 0.000, C 0.000 }
gfCNCPoint1[28793] = {X 236.1733, Y 101.3775, Z -2.1667, A 0.000, B 0.000, C 0.000 }
gfCNCPoint1[28794] = {X 235.3542, Y 101.8922, Z -2.1667, A 0.000, B 0.000, C 0.000 }
gfCNCPoint1[28795] = {X 234.4411, Y 102.2117, Z -2.1667, A 0.000, B 0.000, C 0.000 }
gfCNCPoint1[28796] = {X 233.4798, Y 102.3200, Z -2.1667, A 0.000, B 0.000, C 0.000 }
gfCNCPoint1[28797] = {X 214.1790, Y 102.3200, Z -2.1667, A 0.000, B 0.000, C 0.000 }
